IF start THEN
FindAndReplace(pSrcString:= ADR(cmdIn), pDeleteString:= ADR('#1#'), pInsertString:= ADR(GVL_HMI.stRecipeInfo.sMethodName), pDstString:= ADR(cmdIn), nDstSize:= SIZEOF(cmdIn));
FindAndReplace(pSrcString:= ADR(cmdIn), pDeleteString:= ADR('#2#'), pInsertString:= ADR(iRevision), pDstString:= ADR(cmdIn), nDstSize:= SIZEOF(cmdIn));
FindAndReplace(pSrcString:= ADR(cmdIn), pDeleteString:= ADR('#3#'), pInsertString:= ADR(GVL_HMI.stRecipeInfo.sCreatedBy), pDstString:= ADR(cmdIn), nDstSize:= SIZEOF(cmdIn));
FindAndReplace(pSrcString:= ADR(cmdIn), pDeleteString:= ADR('#4#'), pInsertString:= ADR(dCreationDate), pDstString:= ADR(cmdIn), nDstSize:= SIZEOF(cmdIn));
FindAndReplace(pSrcString:= ADR(cmdIn), pDeleteString:= ADR('#5#'), pInsertString:= ADR(Rinse1), pDstString:= ADR(cmdIn), nDstSize:= SIZEOF(cmdIn));
FindAndReplace(pSrcString:= ADR(cmdIn), pDeleteString:= ADR('#6#'), pInsertString:= ADR(Rinse2), pDstString:= ADR(cmdIn), nDstSize:= SIZEOF(cmdIn));
FindAndReplace(pSrcString:= ADR(cmdIn), pDeleteString:= ADR('#7#'), pInsertString:= ADR(Wash1), pDstString:= ADR(cmdIn), nDstSize:= SIZEOF(cmdIn));
FindAndReplace(pSrcString:= ADR(cmdIn), pDeleteString:= ADR('#8#'), pInsertString:= ADR(Wash2), pDstString:= ADR(cmdIn), nDstSize:= SIZEOF(cmdIn));
FindAndReplace(pSrcString:= ADR(cmdIn), pDeleteString:= ADR('#9#'), pInsertString:= ADR(Rinse12), pDstString:= ADR(cmdIn), nDstSize:= SIZEOF(cmdIn));
FindAndReplace(pSrcString:= ADR(cmdIn), pDeleteString:= ADR('#10#'), pInsertString:= ADR(Rinse22), pDstString:= ADR(cmdIn), nDstSize:= SIZEOF(cmdIn));
FindAndReplace(pSrcString:= ADR(cmdIn), pDeleteString:= ADR('#11#'), pInsertString:= ADR(Wash12), pDstString:= ADR(cmdIn), nDstSize:= SIZEOF(cmdIn));
FindAndReplace(pSrcString:= ADR(cmdIn), pDeleteString:= ADR('#12#'), pInsertString:= ADR(Wash22), pDstString:= ADR(cmdIn), nDstSize:= SIZEOF(cmdIn));
FindAndReplace(pSrcString:= ADR(cmdIn), pDeleteString:= ADR('#13#'), pInsertString:= ADR(Rinse13), pDstString:= ADR(cmdIn), nDstSize:= SIZEOF(cmdIn));
FindAndReplace(pSrcString:= ADR(cmdIn), pDeleteString:= ADR('#14#'), pInsertString:= ADR(Rinse23), pDstString:= ADR(cmdIn), nDstSize:= SIZEOF(cmdIn));
FindAndReplace(pSrcString:= ADR(cmdIn), pDeleteString:= ADR('#15#'), pInsertString:= ADR(Wash13), pDstString:= ADR(cmdIn), nDstSize:= SIZEOF(cmdIn));
FindAndReplace(pSrcString:= ADR(cmdIn), pDeleteString:= ADR('#16#'), pInsertString:= ADR(Wash23), pDstString:= ADR(cmdIn), nDstSize:= SIZEOF(cmdIn));
FindAndReplace(pSrcString:= ADR(cmdIn), pDeleteString:= ADR('#17#'), pInsertString:= ADR(soakTime), pDstString:= ADR(cmdIn), nDstSize:= SIZEOF(cmdIn));
FindAndReplace(pSrcString:= ADR(cmdIn), pDeleteString:= ADR('#18#'), pInsertString:= ADR(agitate_1_Time), pDstString:= ADR(cmdIn), nDstSize:= SIZEOF(cmdIn));
FindAndReplace(pSrcString:= ADR(cmdIn), pDeleteString:= ADR('#19#'), pInsertString:= ADR(agitate_2_Time), pDstString:= ADR(cmdIn), nDstSize:= SIZEOF(cmdIn));
FindAndReplace(pSrcString:= ADR(cmdIn), pDeleteString:= ADR('#20#'), pInsertString:= ADR(vialsToFill), pDstString:= ADR(cmdIn), nDstSize:= SIZEOF(cmdIn));
FindAndReplace(pSrcString:= ADR(cmdIn), pDeleteString:= ADR('#21#'), pInsertString:= ADR(vialPrimeVol), pDstString:= ADR(cmdIn), nDstSize:= SIZEOF(cmdIn));
FindAndReplace(pSrcString:= ADR(cmdIn), pDeleteString:= ADR('#22#'), pInsertString:= ADR(vial_1_FillVol), pDstString:= ADR(cmdIn), nDstSize:= SIZEOF(cmdIn));
FindAndReplace(pSrcString:= ADR(cmdIn), pDeleteString:= ADR('#23#'), pInsertString:= ADR(vial_2_4_FillVol), pDstString:= ADR(cmdIn), nDstSize:= SIZEOF(cmdIn));
FindAndReplace(pSrcString:= ADR(cmdIn), pDeleteString:= ADR('#24#'), pInsertString:= ADR(airDryTime), pDstString:= ADR(cmdIn), nDstSize:= SIZEOF(cmdIn));
FindAndReplace(pSrcString:= ADR(cmdIn), pDeleteString:= ADR('#25#'), pInsertString:= ADR('activated'), pDstString:= ADR(cmdIn), nDstSize:= SIZEOF(cmdIn));

END_IF
END_METHOD

METHOD insertRunValues : BOOL
VAR_INPUT
	start: bool;
END_VAR

VAR
	methodID: STRING;
	CalibrationNo: STRING;
END_VAR
methodID:= INT_TO_STRING(GVL_DB.stPostRunInfo.methodID);
CalibrationNo:= INT_TO_STRING(GVL_DB.stPostRunInfo.CalibrationNo);

IF start THEN
FindAndReplace(pSrcString:= ADR(cmdIn), pDeleteString:= ADR('#1#'), pInsertString:= ADR(GVL_DB.stPostRunInfo.analyst), pDstString:= ADR(cmdIn), nDstSize:= SIZEOF(cmdIn));
FindAndReplace(pSrcString:= ADR(cmdIn), pDeleteString:= ADR('#2#'), pInsertString:= ADR(GVL_DB.stPostRunInfo.comment), pDstString:= ADR(cmdIn), nDstSize:= SIZEOF(cmdIn));
FindAndReplace(pSrcString:= ADR(cmdIn), pDeleteString:= ADR('#3#'), pInsertString:= ADR(GVL_DB.stPostRunInfo.softwareVersion), pDstString:= ADR(cmdIn), nDstSize:= SIZEOF(cmdIn));
FindAndReplace(pSrcString:= ADR(cmdIn), pDeleteString:= ADR('#4#'), pInsertString:= ADR(GVL_DB.stPostRunInfo.sysMasterRevision), pDstString:= ADR(cmdIn), nDstSize:= SIZEOF(cmdIn));
FindAndReplace(pSrcString:= ADR(cmdIn), pDeleteString:= ADR('#5#'), pInsertString:= ADR(GVL_DB.stPostRunInfo.sysSettingsRevision), pDstString:= ADR(cmdIn), nDstSize:= SIZEOF(cmdIn));
FindAndReplace(pSrcString:= ADR(cmdIn), pDeleteString:= ADR('#6#'), pInsertString:= ADR(GVL_DB.stPostRunInfo.meterVelocity), pDstString:= ADR(cmdIn), nDstSize:= SIZEOF(cmdIn));
FindAndReplace(pSrcString:= ADR(cmdIn), pDeleteString:= ADR('#7#'), pInsertString:= ADR(GVL_DB.stPostRunInfo.runVelocity), pDstString:= ADR(cmdIn), nDstSize:= SIZEOF(cmdIn));
FindAndReplace(pSrcString:= ADR(cmdIn), pDeleteString:= ADR('#8#'), pInsertString:= ADR(GVL_DB.stPostRunInfo.emptyTubesFactor), pDstString:= ADR(cmdIn), nDstSize:= SIZEOF(cmdIn));
FindAndReplace(pSrcString:= ADR(cmdIn), pDeleteString:= ADR('#9#'), pInsertString:= ADR(GVL_DB.stPostRunInfo.fillTubesFactor), pDstString:= ADR(cmdIn), nDstSize:= SIZEOF(cmdIn));
FindAndReplace(pSrcString:= ADR(cmdIn), pDeleteString:= ADR('#10#'), pInsertString:= ADR(GVL_DB.stPostRunInfo.solvent1NameRevision), pDstString:= ADR(cmdIn), nDstSize:= SIZEOF(cmdIn));
FindAndReplace(pSrcString:= ADR(cmdIn), pDeleteString:= ADR('#11#'), pInsertString:= ADR(GVL_DB.stPostRunInfo.solvent2NameRevision), pDstString:= ADR(cmdIn), nDstSize:= SIZEOF(cmdIn));
FindAndReplace(pSrcString:= ADR(cmdIn), pDeleteString:= ADR('#12#'), pInsertString:= ADR(GVL_DB.stPostRunInfo.solvent3NameRevision), pDstString:= ADR(cmdIn), nDstSize:= SIZEOF(cmdIn));
FindAndReplace(pSrcString:= ADR(cmdIn), pDeleteString:= ADR('#13#'), pInsertString:= ADR(GVL_DB.stPostRunInfo.solvent4NameRevision), pDstString:= ADR(cmdIn), nDstSize:= SIZEOF(cmdIn));
FindAndReplace(pSrcString:= ADR(cmdIn), pDeleteString:= ADR('#14#'), pInsertString:= ADR(GVL_DB.stPostRunInfo.timeEventStarted), pDstString:= ADR(cmdIn), nDstSize:= SIZEOF(cmdIn));
FindAndReplace(pSrcString:= ADR(cmdIn), pDeleteString:= ADR('#15#'), pInsertString:= ADR(GVL_DB.stPostRunInfo.timeEventCompleted), pDstString:= ADR(cmdIn), nDstSize:= SIZEOF(cmdIn));
FindAndReplace(pSrcString:= ADR(cmdIn), pDeleteString:= ADR('#16#'), pInsertString:= ADR(methodID), pDstString:= ADR(cmdIn), nDstSize:= SIZEOF(cmdIn));
FindAndReplace(pSrcString:= ADR(cmdIn), pDeleteString:= ADR('#17#'), pInsertString:= ADR(CalibrationNo), pDstString:= ADR(cmdIn), nDstSize:= SIZEOF(cmdIn));
END_IF
END_METHOD

METHOD insertSolvent : BOOL
VAR_INPUT
	start: BOOL;
END_VAR


VAR

END_VAR


IF start THEN
	FindAndReplace(pSrcString:= ADR(cmdIn), pDeleteString:= ADR('#1#'), pInsertString:= ADR(GVL_DB.stSolvents.solventName1), pDstString:= ADR(cmdIn), nDstSize:= SIZEOF(cmdIn));
	FindAndReplace(pSrcString:= ADR(cmdIn), pDeleteString:= ADR('#2#'), pInsertString:= ADR(GVL_DB.stSolvents.solventName2), pDstString:= ADR(cmdIn), nDstSize:= SIZEOF(cmdIn));
	FindAndReplace(pSrcString:= ADR(cmdIn), pDeleteString:= ADR('#3#'), pInsertString:= ADR(GVL_DB.stSolvents.solventName3), pDstString:= ADR(cmdIn), nDstSize:= SIZEOF(cmdIn));
	FindAndReplace(pSrcString:= ADR(cmdIn), pDeleteString:= ADR('#4#'), pInsertString:= ADR(GVL_DB.stSolvents.solventName4), pDstString:= ADR(cmdIn), nDstSize:= SIZEOF(cmdIn));
	FindAndReplace(pSrcString:= ADR(cmdIn), pDeleteString:= ADR('#5#'), pInsertString:= ADR(GVL_DB.stSolvents.density1), pDstString:= ADR(cmdIn), nDstSize:= SIZEOF(cmdIn));
	FindAndReplace(pSrcString:= ADR(cmdIn), pDeleteString:= ADR('#6#'), pInsertString:= ADR(GVL_DB.stSolvents.density2), pDstString:= ADR(cmdIn), nDstSize:= SIZEOF(cmdIn));
	FindAndReplace(pSrcString:= ADR(cmdIn), pDeleteString:= ADR('#7#'), pInsertString:= ADR(GVL_DB.stSolvents.density3), pDstString:= ADR(cmdIn), nDstSize:= SIZEOF(cmdIn));
	FindAndReplace(pSrcString:= ADR(cmdIn), pDeleteString:= ADR('#8#'), pInsertString:= ADR(GVL_DB.stSolvents.density4), pDstString:= ADR(cmdIn), nDstSize:= SIZEOF(cmdIn));
	FindAndReplace(pSrcString:= ADR(cmdIn), pDeleteString:= ADR('#9#'), pInsertString:= ADR(GVL_DB.stSolvents.addedBy), pDstString:= ADR(cmdIn), nDstSize:= SIZEOF(cmdIn));
	FindAndReplace(pSrcString:= ADR(cmdIn), pDeleteString:= ADR('#10#'), pInsertString:= ADR(GVL_DB.stSolvents.addedDate), pDstString:= ADR(cmdIn), nDstSize:= SIZEOF(cmdIn));
END_IF
END_METHOD

METHOD insertSys : BOOL
VAR_INPUT
	start: BOOL;
END_VAR

VAR
	bGeneralSealAndPump: STRING;
	rAcceptanceCriteria: STRING;
	iAllowableFailures: STRING;
	iReplicatesSetpoint: STRING;
	iCalIntervalDays: STRING;
	iAirDryTimeSec: STRING;
	iAllowableLeakTestFailures: STRING;
	tLeakTestBuildUpTime: STRING;
	tLeakTestMonitorTime: STRING;
	rLeakTestPressureLimit: STRING;
	sealPosition: STRING;
	dryposition: STRING;
	rM1Velocity: STRING;
	iMeterVelocity: STRING;
	iRunVelocity: STRING;
	iEmptyFactor: STRING;
	iFillolventTubesFactor: STRING;
	abovecalibration: STRING;
	vialsetspacing: STRING;
	intoresbottom: STRING;
	intodispense: STRING;
	intoweight: STRING;
	intovials: STRING;
	bDisplayManualControl: STRING;
	bCheckLogonEachRun: STRING;
	abovevialset1: STRING;
	intoWaste: STRING;
	userName: STRING;
	savedDate: STRING;
	
	// Timestamp generation (local system time)
    fbLocalSystemTime : FB_LocalSystemTime;
    stLocal           : TIMESTRUCT;
    sStamp            : STRING(32);
    sHH               : STRING(2);
    sMM               : STRING(2);
    sSS               : STRING(2);
    sMMo              : STRING(3);
    sDD               : STRING(2);
	bDTReady		  : BOOL := FALSE;

END_VAR
bGeneralSealAndPump := BOOL_TO_STRING(GVL_Settings.bGeneralSealAndPump);
rAcceptanceCriteria := LREAL_TO_STRING(GVL_Settings.stCalibParameters.rAcceptanceCriteria);
iAllowableFailures  := USINT_TO_STRING(GVL_Settings.stCalibParameters.iAllowableFailures);
iReplicatesSetpoint := UINT_TO_STRING(GVL_Settings.stCalibParameters.iReplicatesSetpoint);
iCalIntervalDays := UINT_TO_STRING(GVL_Settings.stCalibParameters.iCalIntervalDays);
iAirDryTimeSec := UINT_TO_STRING(GVL_Settings.stCalibParameters.iAirDryTimeSec);
iAllowableLeakTestFailures := UINT_TO_STRING(GVL_Settings.stLeakTestParameters.iAllowableLeakTestFailures);
tLeakTestBuildUpTime := UINT_TO_STRING(GVL_Settings.stLeakTestParameters.tLeakTestBuildUpTime);
tLeakTestMonitorTime := UINT_TO_STRING(GVL_Settings.stLeakTestParameters.tLeakTestMonitorTime);
rLeakTestPressureLimit := REAL_TO_STRING(GVL_Settings.stLeakTestParameters.rLeakTestPressureLimit);
sealPosition := INT_TO_STRING(GVL_Settings.stMachineParam.aM1Position[2]);
dryposition := INT_TO_STRING(GVL_Settings.stMachineParam.aM1Position[3]);
rM1Velocity := LREAL_TO_STRING(GVL_Settings.stMachineParam.rM1Velocity);
iMeterVelocity := UINT_TO_STRING(GVL_Settings.stPumpParameters.iMeterVelocity);
iRunVelocity := UINT_TO_STRING(GVL_Settings.stPumpParameters.iRunVelocity);
iEmptyFactor := UINT_TO_STRING(GVL_Settings.stPumpParameters.iEmptyFactor);
iFillolventTubesFactor := UINT_TO_STRING(GVL_Settings.stPumpParameters.iFillolventTubesFactor);
abovecalibration := INT_TO_STRING(GVL_Settings.stMachineParam.aM3Position[4]);
vialsetspacing := INT_TO_STRING(GVL_Settings.stMachineParam.aM3Position[3]);
intoresbottom := INT_TO_STRING(GVL_Settings.stMachineParam.aM2Position[4]);
intodispense := INT_TO_STRING(GVL_Settings.stMachineParam.aM2Position[5]);
intoweight := INT_TO_STRING(GVL_Settings.stMachineParam.aM2Position[6]);
intovials := INT_TO_STRING(GVL_Settings.stMachineParam.aM2Position[3]);
bDisplayManualControl := BOOL_TO_STRING(GVL_Settings.bDisplayManualControl);
bCheckLogonEachRun := BOOL_TO_STRING(GVL_Settings.bCheckLogonEachRun);
abovevialset1 := INT_TO_STRING(GVL_Settings.stMachineParam.aM3Position[2]);
intoWaste := INT_TO_STRING(GVL_Settings.stMachineParam.aM2Position[2]);
userName := GVL_HMI.sUserNameEventTriggered;
savedDate := GVL_HMI.sDateAndTimeEventTriggered;

IF start THEN
	FindAndReplace(pSrcString:= ADR(cmdIn), pDeleteString:= ADR('#1#'), pInsertString:= ADR(bGeneralSealAndPump), pDstString:= ADR(cmdIn), nDstSize:= SIZEOF(cmdIn));
	FindAndReplace(pSrcString:= ADR(cmdIn), pDeleteString:= ADR('#2#'), pInsertString:= ADR(rAcceptanceCriteria), pDstString:= ADR(cmdIn), nDstSize:= SIZEOF(cmdIn));
	FindAndReplace(pSrcString:= ADR(cmdIn), pDeleteString:= ADR('#3#'), pInsertString:= ADR(iAllowableFailures), pDstString:= ADR(cmdIn), nDstSize:= SIZEOF(cmdIn));
	FindAndReplace(pSrcString:= ADR(cmdIn), pDeleteString:= ADR('#4#'), pInsertString:= ADR(iReplicatesSetpoint), pDstString:= ADR(cmdIn), nDstSize:= SIZEOF(cmdIn));
	FindAndReplace(pSrcString:= ADR(cmdIn), pDeleteString:= ADR('#5#'), pInsertString:= ADR(iCalIntervalDays), pDstString:= ADR(cmdIn), nDstSize:= SIZEOF(cmdIn));
	FindAndReplace(pSrcString:= ADR(cmdIn), pDeleteString:= ADR('#6#'), pInsertString:= ADR('N/A'), pDstString:= ADR(cmdIn), nDstSize:= SIZEOF(cmdIn));
	FindAndReplace(pSrcString:= ADR(cmdIn), pDeleteString:= ADR('#7#'), pInsertString:= ADR(iAirDryTimeSec), pDstString:= ADR(cmdIn), nDstSize:= SIZEOF(cmdIn));
	FindAndReplace(pSrcString:= ADR(cmdIn), pDeleteString:= ADR('#8#'), pInsertString:= ADR(iAllowableLeakTestFailures), pDstString:= ADR(cmdIn), nDstSize:= SIZEOF(cmdIn));
	FindAndReplace(pSrcString:= ADR(cmdIn), pDeleteString:= ADR('#9#'), pInsertString:= ADR(tLeakTestBuildUpTime), pDstString:= ADR(cmdIn), nDstSize:= SIZEOF(cmdIn));
	FindAndReplace(pSrcString:= ADR(cmdIn), pDeleteString:= ADR('#10#'), pInsertString:= ADR(tLeakTestMonitorTime), pDstString:= ADR(cmdIn), nDstSize:= SIZEOF(cmdIn));
	FindAndReplace(pSrcString:= ADR(cmdIn), pDeleteString:= ADR('#11#'), pInsertString:= ADR(rLeakTestPressureLimit), pDstString:= ADR(cmdIn), nDstSize:= SIZEOF(cmdIn));
	FindAndReplace(pSrcString:= ADR(cmdIn), pDeleteString:= ADR('#12#'), pInsertString:= ADR(sealPosition), pDstString:= ADR(cmdIn), nDstSize:= SIZEOF(cmdIn));
	FindAndReplace(pSrcString:= ADR(cmdIn), pDeleteString:= ADR('#13#'), pInsertString:= ADR(dryposition), pDstString:= ADR(cmdIn), nDstSize:= SIZEOF(cmdIn));
	FindAndReplace(pSrcString:= ADR(cmdIn), pDeleteString:= ADR('#14#'), pInsertString:= ADR(rM1Velocity), pDstString:= ADR(cmdIn), nDstSize:= SIZEOF(cmdIn));
	FindAndReplace(pSrcString:= ADR(cmdIn), pDeleteString:= ADR('#15#'), pInsertString:= ADR('N/A'), pDstString:= ADR(cmdIn), nDstSize:= SIZEOF(cmdIn));
	FindAndReplace(pSrcString:= ADR(cmdIn), pDeleteString:= ADR('#16#'), pInsertString:= ADR('N/A'), pDstString:= ADR(cmdIn), nDstSize:= SIZEOF(cmdIn));
	FindAndReplace(pSrcString:= ADR(cmdIn), pDeleteString:= ADR('#17#'), pInsertString:= ADR('N/A'), pDstString:= ADR(cmdIn), nDstSize:= SIZEOF(cmdIn));
	FindAndReplace(pSrcString:= ADR(cmdIn), pDeleteString:= ADR('#18#'), pInsertString:= ADR(iMeterVelocity), pDstString:= ADR(cmdIn), nDstSize:= SIZEOF(cmdIn));
	FindAndReplace(pSrcString:= ADR(cmdIn), pDeleteString:= ADR('#19#'), pInsertString:= ADR(iRunVelocity), pDstString:= ADR(cmdIn), nDstSize:= SIZEOF(cmdIn));
	FindAndReplace(pSrcString:= ADR(cmdIn), pDeleteString:= ADR('#20#'), pInsertString:= ADR(iEmptyFactor), pDstString:= ADR(cmdIn), nDstSize:= SIZEOF(cmdIn));
	FindAndReplace(pSrcString:= ADR(cmdIn), pDeleteString:= ADR('#21#'), pInsertString:= ADR(iFillolventTubesFactor), pDstString:= ADR(cmdIn), nDstSize:= SIZEOF(cmdIn));
	FindAndReplace(pSrcString:= ADR(cmdIn), pDeleteString:= ADR('#22#'), pInsertString:= ADR(abovecalibration), pDstString:= ADR(cmdIn), nDstSize:= SIZEOF(cmdIn));
	FindAndReplace(pSrcString:= ADR(cmdIn), pDeleteString:= ADR('#23#'), pInsertString:= ADR(vialsetspacing), pDstString:= ADR(cmdIn), nDstSize:= SIZEOF(cmdIn));
	FindAndReplace(pSrcString:= ADR(cmdIn), pDeleteString:= ADR('#24#'), pInsertString:= ADR(intoresbottom), pDstString:= ADR(cmdIn), nDstSize:= SIZEOF(cmdIn));
	FindAndReplace(pSrcString:= ADR(cmdIn), pDeleteString:= ADR('#25#'), pInsertString:= ADR(intodispense), pDstString:= ADR(cmdIn), nDstSize:= SIZEOF(cmdIn));
	FindAndReplace(pSrcString:= ADR(cmdIn), pDeleteString:= ADR('#26#'), pInsertString:= ADR(intoweight), pDstString:= ADR(cmdIn), nDstSize:= SIZEOF(cmdIn));
	FindAndReplace(pSrcString:= ADR(cmdIn), pDeleteString:= ADR('#27#'), pInsertString:= ADR(intovials), pDstString:= ADR(cmdIn), nDstSize:= SIZEOF(cmdIn));
	FindAndReplace(pSrcString:= ADR(cmdIn), pDeleteString:= ADR('#28#'), pInsertString:= ADR(bDisplayManualControl), pDstString:= ADR(cmdIn), nDstSize:= SIZEOF(cmdIn));
	FindAndReplace(pSrcString:= ADR(cmdIn), pDeleteString:= ADR('#29#'), pInsertString:= ADR(bCheckLogonEachRun), pDstString:= ADR(cmdIn), nDstSize:= SIZEOF(cmdIn));
	FindAndReplace(pSrcString:= ADR(cmdIn), pDeleteString:= ADR('#30#'), pInsertString:= ADR(userName), pDstString:= ADR(cmdIn), nDstSize:= SIZEOF(cmdIn));
	FindAndReplace(pSrcString:= ADR(cmdIn), pDeleteString:= ADR('#31#'), pInsertString:= ADR(savedDate), pDstString:= ADR(cmdIn), nDstSize:= SIZEOF(cmdIn));
	FindAndReplace(pSrcString:= ADR(cmdIn), pDeleteString:= ADR('#32#'), pInsertString:= ADR(abovevialset1), pDstString:= ADR(cmdIn), nDstSize:= SIZEOF(cmdIn));
	FindAndReplace(pSrcString:= ADR(cmdIn), pDeleteString:= ADR('#33#'), pInsertString:= ADR(intoWaste), pDstString:= ADR(cmdIn), nDstSize:= SIZEOF(cmdIn));
END_IF
END_METHOD

METHOD insertUser : BOOL
VAR_INPUT
	start: BOOL;
	line: INT;
END_VAR


IF start THEN
	FindAndReplace(pSrcString:= ADR(cmdIn), pDeleteString:= ADR('#1#'), pInsertString:= ADR(GVL_DB.astData_CUL[line].userID), pDstString:= ADR(cmdIn), nDstSize:= SIZEOF(cmdIn));
	FindAndReplace(pSrcString:= ADR(cmdIn), pDeleteString:= ADR('#2#'), pInsertString:= ADR(GVL_DB.astData_CUL[line].acessLevel), pDstString:= ADR(cmdIn), nDstSize:= SIZEOF(cmdIn));
	FindAndReplace(pSrcString:= ADR(cmdIn), pDeleteString:= ADR('#3#'), pInsertString:= ADR(GVL_DB.astData_CUL[line].transactionType), pDstString:= ADR(cmdIn), nDstSize:= SIZEOF(cmdIn));
	FindAndReplace(pSrcString:= ADR(cmdIn), pDeleteString:= ADR('#4#'), pInsertString:= ADR(GVL_DB.astData_CUL[line].transactionDate), pDstString:= ADR(cmdIn), nDstSize:= SIZEOF(cmdIn));
	FindAndReplace(pSrcString:= ADR(cmdIn), pDeleteString:= ADR('#5#'), pInsertString:= ADR(GVL_DB.astData_CUL[line].transactedBy), pDstString:= ADR(cmdIn), nDstSize:= SIZEOF(cmdIn));
	FindAndReplace(pSrcString:= ADR(cmdIn), pDeleteString:= ADR('#6#'), pInsertString:= ADR(GVL_DB.astData_CUL[line].addDate), pDstString:= ADR(cmdIn), nDstSize:= SIZEOF(cmdIn));
	FindAndReplace(pSrcString:= ADR(cmdIn), pDeleteString:= ADR('#7#'), pInsertString:= ADR(GVL_DB.astData_CUL[line].enteredBy), pDstString:= ADR(cmdIn), nDstSize:= SIZEOF(cmdIn));
END_IF
END_METHOD

METHOD insertUserMgmtHistory : BOOL
VAR_INPUT
	start : BOOL := FALSE;
END_VAR
VAR
    sOldAutoLogoutMin : STRING(20);
    sNewAutoLogoutMin : STRING(20);
END_VAR
sOldAutoLogoutMin := INT_TO_STRING(GVL_HMI.stUserMgmtHistoryEvent.iOldAutoLogoutMin);
sNewAutoLogoutMin := INT_TO_STRING(GVL_HMI.stUserMgmtHistoryEvent.iNewAutoLogoutMin);

IF start THEN

    FindAndReplace(
        pSrcString := ADR(cmdIn), 
        pDeleteString := ADR('#1#'), 
        pInsertString := ADR(GVL_HMI.stUserMgmtHistoryEvent.sTargetUser), 
        pDstString := ADR(cmdIn), 
        nDstSize := SIZEOF(cmdIn)
    );

    FindAndReplace(
        pSrcString := ADR(cmdIn), 
        pDeleteString := ADR('#2#'), 
        pInsertString := ADR(GVL_HMI.stUserMgmtHistoryEvent.sEventType), 
        pDstString := ADR(cmdIn), 
        nDstSize := SIZEOF(cmdIn)
    );

    FindAndReplace(
        pSrcString := ADR(cmdIn), 
        pDeleteString := ADR('#3#'), 
        pInsertString := ADR(GVL_HMI.stUserMgmtHistoryEvent.sOldGroup), 
        pDstString := ADR(cmdIn), 
        nDstSize := SIZEOF(cmdIn)
    );

    FindAndReplace(
        pSrcString := ADR(cmdIn), 
        pDeleteString := ADR('#4#'), 
        pInsertString := ADR(GVL_HMI.stUserMgmtHistoryEvent.sNewGroup), 
        pDstString := ADR(cmdIn), 
        nDstSize := SIZEOF(cmdIn)
    );

    FindAndReplace(
        pSrcString := ADR(cmdIn), 
        pDeleteString := ADR('#5#'), 
        pInsertString := ADR(sOldAutoLogoutMin), 
        pDstString := ADR(cmdIn), 
        nDstSize := SIZEOF(cmdIn)
    );

    FindAndReplace(
        pSrcString := ADR(cmdIn), 
        pDeleteString := ADR('#6#'), 
        pInsertString := ADR(sNewAutoLogoutMin), 
        pDstString := ADR(cmdIn), 
        nDstSize := SIZEOF(cmdIn)
    );

    FindAndReplace(
        pSrcString := ADR(cmdIn), 
        pDeleteString := ADR('#7#'), 
        pInsertString := ADR(GVL_HMI.stUserMgmtHistoryEvent.sPerformedBy), 
        pDstString := ADR(cmdIn), 
        nDstSize := SIZEOF(cmdIn)
    );

    FindAndReplace(
        pSrcString := ADR(cmdIn), 
        pDeleteString := ADR('#8#'), 
        pInsertString := ADR(GVL_HMI.stUserMgmtHistoryEvent.sSourceScreen), 
        pDstString := ADR(cmdIn), 
        nDstSize := SIZEOF(cmdIn)
    );

    FindAndReplace(
        pSrcString := ADR(cmdIn), 
        pDeleteString := ADR('#9#'), 
        pInsertString := ADR(GVL_HMI.stUserMgmtHistoryEvent.sEventComment), 
        pDstString := ADR(cmdIn), 
        nDstSize := SIZEOF(cmdIn)
    );

END_IF
END_METHOD

METHOD insertVD : BOOL
VAR_INPUT
	start: BOOL;
	methodID: STRING;
	line: INT;
END_VAR


VAR
	sysRevisionNo: STRING;
END_VAR


IF start THEN
	FindAndReplace(pSrcString:= ADR(cmdIn), pDeleteString:= ADR('#1#'), pInsertString:= ADR(GVL_DB.astVolData[line].pump), pDstString:= ADR(cmdIn), nDstSize:= SIZEOF(cmdIn));
	FindAndReplace(pSrcString:= ADR(cmdIn), pDeleteString:= ADR('#2#'), pInsertString:= ADR(GVL_DB.astVolData[line].stage), pDstString:= ADR(cmdIn), nDstSize:= SIZEOF(cmdIn));
	FindAndReplace(pSrcString:= ADR(cmdIn), pDeleteString:= ADR('#3#'), pInsertString:= ADR(GVL_DB.astVolData[line].rinse1), pDstString:= ADR(cmdIn), nDstSize:= SIZEOF(cmdIn));
	FindAndReplace(pSrcString:= ADR(cmdIn), pDeleteString:= ADR('#4#'), pInsertString:= ADR(GVL_DB.astVolData[line].rinse2), pDstString:= ADR(cmdIn), nDstSize:= SIZEOF(cmdIn));
	FindAndReplace(pSrcString:= ADR(cmdIn), pDeleteString:= ADR('#5#'), pInsertString:= ADR(GVL_DB.astVolData[line].wash1), pDstString:= ADR(cmdIn), nDstSize:= SIZEOF(cmdIn));
	FindAndReplace(pSrcString:= ADR(cmdIn), pDeleteString:= ADR('#6#'), pInsertString:= ADR(GVL_DB.astVolData[line].wash2), pDstString:= ADR(cmdIn), nDstSize:= SIZEOF(cmdIn));
	FindAndReplace(pSrcString:= ADR(cmdIn), pDeleteString:= ADR('#7#'), pInsertString:= ADR(methodID), pDstString:= ADR(cmdIn), nDstSize:= SIZEOF(cmdIn));
END_IF
END_METHOD

METHOD selectCalibHeader : BOOL
VAR_INPUT
	start : BOOL;
    calibrationNo : STRING;
END_VAR
IF start THEN
    FindAndReplace(
        pSrcString := ADR(cmdSlc),
        pDeleteString := ADR('#1#'),
        pInsertString := ADR(calibrationNo),
        pDstString := ADR(cmdSlc),
        nDstSize := SIZEOF(cmdSlc)
    );
END_IF
END_METHOD

METHOD selectCalibReportHeaderByID : BOOL
VAR_INPUT
	start         : BOOL;
    calibrationID : STRING;
END_VAR
IF start THEN
    Clear_PumpCalibReportBuffers();
    cmdSlc := GVL_DB.slctPumpCalibHeaderByNo1;

    FindAndReplace(
        pSrcString:= ADR(cmdSlc),
        pDeleteString:= ADR('#1#'),
        pInsertString:= ADR(calibrationID),
        pDstString:= ADR(cmdSlc),
        nDstSize:= SIZEOF(cmdSlc)
    );
END_IF
END_METHOD

METHOD selectCalibReportListByDate : BOOL
VAR_INPUT
	start    : BOOL;
    dateFrom : STRING;
    dateTo   : STRING;
END_VAR
IF start THEN
    cmdSlc := GVL_DB.slctCalibReportListByDate;

    FindAndReplace(
        pSrcString    := ADR(cmdSlc),
        pDeleteString := ADR('#1#'),
        pInsertString := ADR(dateFrom),
        pDstString    := ADR(cmdSlc),
        nDstSize      := SIZEOF(cmdSlc)
    );

    FindAndReplace(
        pSrcString    := ADR(cmdSlc),
        pDeleteString := ADR('#2#'),
        pInsertString := ADR(dateTo),
        pDstString    := ADR(cmdSlc),
        nDstSize      := SIZEOF(cmdSlc)
    );
END_IF
END_METHOD

METHOD selectCalibReportValuesByID : BOOL
VAR_INPUT
	start         : BOOL;
    calibrationID : STRING;
END_VAR
IF start THEN
    cmdSlc := GVL_DB.slctPumpCalibValuesByNo1;

    FindAndReplace(
        pSrcString:= ADR(cmdSlc),
        pDeleteString:= ADR('#1#'),
        pInsertString:= ADR(calibrationID),
        pDstString:= ADR(cmdSlc),
        nDstSize:= SIZEOF(cmdSlc)
    );
END_IF
END_METHOD

METHOD selectLinearByID : BOOL
VAR_INPUT
	start    : BOOL;
    linearID : STRING;
END_VAR
IF start THEN
    IF linearID = '' THEN
        cmdSlc := '';
        RETURN;
    END_IF

    cmdSlc := GVL_DB.slctLinearByID;

    FindAndReplace(
        pSrcString := ADR(cmdSlc),
        pDeleteString := ADR('#1#'),
        pInsertString := ADR(linearID),
        pDstString := ADR(cmdSlc),
        nDstSize := SIZEOF(cmdSlc)
    );
END_IF
END_METHOD

METHOD selectLinearReportSearchByDate : BOOL
VAR_INPUT
	start    : BOOL;
    dateFrom : STRING;
    dateTo   : STRING;
END_VAR
IF start THEN
    cmdSlc := GVL_DB.slctLinearReportListByDate;

    FindAndReplace(
        pSrcString := ADR(cmdSlc),
        pDeleteString := ADR('#1#'),
        pInsertString := ADR(dateFrom),
        pDstString := ADR(cmdSlc),
        nDstSize := SIZEOF(cmdSlc)
    );

    FindAndReplace(
        pSrcString := ADR(cmdSlc),
        pDeleteString := ADR('#2#'),
        pInsertString := ADR(dateTo),
        pDstString := ADR(cmdSlc),
        nDstSize := SIZEOF(cmdSlc)
    );
END_IF
END_METHOD

METHOD selectMethod : BOOL
VAR_INPUT
	start: BOOL;
	methodName: STRING;
	methodRevision: STRING;
END_VAR

IF start THEN
FindAndReplace(pSrcString:= ADR(cmdSlc), pDeleteString:= ADR('#1#'), pInsertString:= ADR(methodName), pDstString:= ADR(cmdSlc), nDstSize:= SIZEOF(cmdSlc));
FindAndReplace(pSrcString:= ADR(cmdSlc), pDeleteString:= ADR('#2#'), pInsertString:= ADR(methodRevision), pDstString:= ADR(cmdSlc), nDstSize:= SIZEOF(cmdSlc));
END_IF
END_METHOD

METHOD selectMethodID : BOOL
VAR_INPUT
	start: BOOL;
	methodName: STRING;
END_VAR

IF start THEN
FindAndReplace(pSrcString:= ADR(cmdSlc), pDeleteString:= ADR('#1#'), pInsertString:= ADR(methodName), pDstString:= ADR(cmdSlc), nDstSize:= SIZEOF(cmdSlc));
END_IF
END_METHOD

METHOD selectMethodReportSearchByDate : BOOL
VAR_INPUT
	start    : BOOL;
	dateFrom : STRING;
	dateTo   : STRING;
END_VAR
// Builds the date-filtered method report search query (latest revision per method).
// Replaces #1# with dateFrom and #2# with dateTo.
IF start THEN
    cmdSlc := GVL_DB.slctMethodReportSearchLatestByDate;

    FindAndReplace(
        pSrcString    := ADR(cmdSlc),
        pDeleteString := ADR('#1#'),
        pInsertString := ADR(dateFrom),
        pDstString    := ADR(cmdSlc),
        nDstSize      := SIZEOF(cmdSlc)
    );

    FindAndReplace(
        pSrcString    := ADR(cmdSlc),
        pDeleteString := ADR('#2#'),
        pInsertString := ADR(dateTo),
        pDstString    := ADR(cmdSlc),
        nDstSize      := SIZEOF(cmdSlc)
    );
END_IF
END_METHOD

METHOD selectPostRunHeaderByID : BOOL
VAR_INPUT
	start : BOOL;
    runID : STRING;
END_VAR
IF start THEN
    cmdSlc := GVL_DB.slctPostRunHeaderByID;

    FindAndReplace(
        pSrcString := ADR(cmdSlc),
        pDeleteString := ADR('#1#'),
        pInsertString := ADR(runID),
        pDstString := ADR(cmdSlc),
        nDstSize := SIZEOF(cmdSlc)
    );
END_IF
END_METHOD

METHOD selectPostRunMethodHeaderByID : BOOL
VAR_INPUT
	start    : BOOL;
    methodID : STRING;
END_VAR
IF start THEN
    cmdSlc := GVL_DB.slctPostRunMethodHeaderByID;

    FindAndReplace(
        pSrcString := ADR(cmdSlc),
        pDeleteString := ADR('#1#'),
        pInsertString := ADR(methodID),
        pDstString := ADR(cmdSlc),
        nDstSize := SIZEOF(cmdSlc)
    );
END_IF
END_METHOD

METHOD selectPostRunVolumeByMethodID : BOOL
VAR_INPUT
	start    : BOOL;
    methodID : STRING;
END_VAR
IF start THEN
    cmdSlc := GVL_DB.slctPostRunVolumeByMethodID;

    FindAndReplace(
        pSrcString := ADR(cmdSlc),
        pDeleteString := ADR('#1#'),
        pInsertString := ADR(methodID),
        pDstString := ADR(cmdSlc),
        nDstSize := SIZEOF(cmdSlc)
    );
END_IF
END_METHOD

METHOD selectRecipeHeaderByID : BOOL
VAR_INPUT
	start    : BOOL;
    methodID : STRING;
END_VAR
IF start THEN
    cmdSlc := GVL_DB.slctMethodHeaderByID;

    FindAndReplace(
        pSrcString := ADR(cmdSlc),
        pDeleteString := ADR('#1#'),
        pInsertString := ADR(methodID),
        pDstString := ADR(cmdSlc),
        nDstSize := SIZEOF(cmdSlc)
    );
END_IF
END_METHOD

METHOD selectRecipeVolumeByID : BOOL
VAR_INPUT
	start    : BOOL;
    methodID : STRING;
END_VAR
IF start THEN
    cmdSlc := GVL_DB.slctMethodVolumeByID;

    FindAndReplace(
        pSrcString := ADR(cmdSlc),
        pDeleteString := ADR('#1#'),
        pInsertString := ADR(methodID),
        pDstString := ADR(cmdSlc),
        nDstSize := SIZEOF(cmdSlc)
    );
END_IF
END_METHOD

METHOD selectSystemSettingsByID : BOOL
VAR_INPUT
	start      : BOOL;
    revisionID : STRING;
END_VAR
IF start THEN
    cmdSlc := GVL_DB.slctSystemSettingsByRevision;

    FindAndReplace(
        pSrcString    := ADR(cmdSlc),
        pDeleteString := ADR('#1#'),
        pInsertString := ADR(revisionID),
        pDstString    := ADR(cmdSlc),
        nDstSize      := SIZEOF(cmdSlc)
    );
END_IF
END_METHOD

METHOD selectSystemSettingsReportLisT : BOOL
VAR_INPUT
	start : BOOL;
END_VAR
IF start THEN
    cmdSlc := GVL_DB.slctSystemSettingsReportList;
END_IF
END_METHOD

METHOD selectSystemSettingsReportListByDate : BOOL
VAR_INPUT
	start    : BOOL;
    dateFrom : STRING;
    dateTo   : STRING;
END_VAR
IF start THEN
    cmdSlc := GVL_DB.slctSystemSettingsReportListByDate;

    FindAndReplace(
        pSrcString    := ADR(cmdSlc),
        pDeleteString := ADR('#1#'),
        pInsertString := ADR(dateFrom),
        pDstString    := ADR(cmdSlc),
        nDstSize      := SIZEOF(cmdSlc)
    );

    FindAndReplace(
        pSrcString    := ADR(cmdSlc),
        pDeleteString := ADR('#2#'),
        pInsertString := ADR(dateTo),
        pDstString    := ADR(cmdSlc),
        nDstSize      := SIZEOF(cmdSlc)
    );
END_IF
END_METHOD

METHOD selectVD : BOOL
VAR_INPUT
	start: BOOL;
	methodID: STRING;
END_VAR

IF start THEN
FindAndReplace(pSrcString:= ADR(cmdSlc), pDeleteString:= ADR('#1#'), pInsertString:= ADR(methodID), pDstString:= ADR(cmdSlc), nDstSize:= SIZEOF(cmdSlc));
END_IF
END_METHOD

METHOD updateMethod : BOOL
VAR_INPUT
	start: BOOL;
	methodName: STRING;
	methodRevision: STRING;
END_VAR

IF start THEN
FindAndReplace(pSrcString:= ADR(cmdIn), pDeleteString:= ADR('#1#'), pInsertString:= ADR(methodName), pDstString:= ADR(cmdIn), nDstSize:= SIZEOF(cmdIn));
FindAndReplace(pSrcString:= ADR(cmdIn), pDeleteString:= ADR('#2#'), pInsertString:= ADR(methodRevision), pDstString:= ADR(cmdIn), nDstSize:= SIZEOF(cmdIn));
END_IF
END_METHOD

END_PROGRAM

// ---- POUs/MARCO/DB/DB_Load_CompleteMethod.TcPOU
PROGRAM DB_Load_CompleteMethod
VAR
	state: INT;
	timer: ton;
	timer2: ton;
	rev: INT := 1;
	x: INT;
END_VAR

VAR_IN_OUT
	start: BOOL;
END_VAR

timer();
timer2();

CASE state OF
	
0:
	IF start THEN
		DB_Query.state:= E_DB_QUERY_STATE.SELECT_WHOLE_METHODS;
		timer(in:=TRUE, pt:=T#1S);
		state:= 10;
	ELSE
		state:= 0;
	END_IF
	
10:

	IF NOT DB_Query.FB_SelectArray.bBusy AND timer.Q THEN
		//start:= TRUE;	
		timer(in:=FALSE);
		GVL_DB.arrCompleteMethod[rev].agitate_1_Time := GVL_DB.stParameter_MR.agitate_1_Time;
		GVL_DB.arrCompleteMethod[rev].agitate_2_Time := GVL_DB.stParameter_MR.agitate_2_Time;
		GVL_DB.arrCompleteMethod[rev].airDryTime := GVL_DB.stParameter_MR.airDryTime;
		GVL_DB.arrCompleteMethod[rev].methodCreatedBy := GVL_DB.stParameter_MR.methodCreatedBy;
		GVL_DB.arrCompleteMethod[rev].methodCreatedOn := GVL_DB.stParameter_MR.methodCreatedOn;
		GVL_DB.arrCompleteMethod[rev].methodID := GVL_DB.stParameter_MR.methodID;
		GVL_DB.arrCompleteMethod[rev].methodName := GVL_DB.stParameter_MR.methodName;
		GVL_DB.arrCompleteMethod[rev].methodRevision := GVL_DB.stParameter_MR.methodRevision;
		GVL_DB.arrCompleteMethod[rev].methodStatus := GVL_DB.stParameter_MR.methodStatus;
		GVL_DB.arrCompleteMethod[rev].soakTime := GVL_DB.stParameter_MR.soakTime;
		GVL_DB.arrCompleteMethod[rev].solvent_R1 := GVL_DB.stParameter_MR.solvent_R1;
		GVL_DB.arrCompleteMethod[rev].solvent_R2 := GVL_DB.stParameter_MR.solvent_R2;
		GVL_DB.arrCompleteMethod[rev].solvent_W1 := GVL_DB.stParameter_MR.solvent_W1;
		GVL_DB.arrCompleteMethod[rev].solvent_W2 := GVL_DB.stParameter_MR.solvent_W2;
		GVL_DB.arrCompleteMethod[rev].time_R1 := GVL_DB.stParameter_MR.time_R1;
		GVL_DB.arrCompleteMethod[rev].time_R2 := GVL_DB.stParameter_MR.time_R2;
		GVL_DB.arrCompleteMethod[rev].time_W1 := GVL_DB.stParameter_MR.time_W1;
		GVL_DB.arrCompleteMethod[rev].time_W2 := GVL_DB.stParameter_MR.time_W2;
		GVL_DB.arrCompleteMethod[rev].velocity_R1 := GVL_DB.stParameter_MR.velocity_R1;
		GVL_DB.arrCompleteMethod[rev].velocity_R2 := GVL_DB.stParameter_MR.velocity_R2;
		GVL_DB.arrCompleteMethod[rev].velocity_W1 := GVL_DB.stParameter_MR.velocity_W1;
		GVL_DB.arrCompleteMethod[rev].velocity_W2 := GVL_DB.stParameter_MR.velocity_W2;
		GVL_DB.arrCompleteMethod[rev].vial_1_FillVol := GVL_DB.stParameter_MR.vial_1_FillVol;
		GVL_DB.arrCompleteMethod[rev].vial_2_4_FillVol := GVL_DB.stParameter_MR.vial_2_4_FillVol;
		GVL_DB.arrCompleteMethod[rev].vialPrimeVol := GVL_DB.stParameter_MR.vialPrimeVol;
		GVL_DB.arrCompleteMethod[rev].vialsToFill := GVL_DB.stParameter_MR.vialsToFill;
		//DB_Query.state:= E_DB_QUERY_STATE.SELECT_VOLUME_DATA;
		timer2(in:= TRUE, pt:= T#5S);
		
		state:= 20;
	ELSE
		state:= 10;
	END_IF
	
20:

	IF NOT DB_Query.FB_SelectArray.bBusy AND timer2.Q THEN
		timer2(in:= FALSE);
		FOR x:= 1 TO 10 BY 1 DO
			GVL_DB.arrCompleteMethod[rev].volumeData[x].pump := GVL_DB.astVolData[x].pump;
			GVL_DB.arrCompleteMethod[rev].volumeData[x].rinse1 := GVL_DB.astVolData[x].rinse1;
			GVL_DB.arrCompleteMethod[rev].volumeData[x].rinse2 := GVL_DB.astVolData[x].rinse2;
			GVL_DB.arrCompleteMethod[rev].volumeData[x].stage := GVL_DB.astVolData[x].stage;
			GVL_DB.arrCompleteMethod[rev].volumeData[x].wash1 := GVL_DB.astVolData[x].wash1;
			GVL_DB.arrCompleteMethod[rev].volumeData[x].wash2 := GVL_DB.astVolData[x].wash2;
			GVL_DB.arrCompleteMethod[rev].volumeData[x].VD_ID := GVL_DB.astVolData[x].VD_ID;
			GVL_DB.arrCompleteMethod[rev].volumeData[x].methodID := GVL_DB.astVolData[x].methodID;
		END_FOR
		DB_Query.state:= E_DB_QUERY_STATE.SELECT_WHOLE_METHODS;
		state:= 30;
	ELSE
		state:= 20;
	END_IF

30:
	IF STRING_TO_INT(GVL_DB.methodRevision) > 1	THEN
		rev:= rev +1;
		GVL_DB.methodRevision:= INT_TO_STRING(STRING_TO_INT(GVL_DB.methodRevision) - 1);
		state:= 0;
	ELSIF STRING_TO_INT(GVL_DB.methodRevision) <= 1 THEN
		start:= FALSE;
		timer(in:= TRUE, pt:= T#5S);
		state:= 40;
	ELSE
		state:= 30;
	END_IF
	
40:
	IF timer.Q THEN
		timer(in:=FALSE);
		rev:= 1;
		state:= 0;
	ELSE
		state:= 40;
	END_IF
END_CASE

END_PROGRAM

// ---- POUs/1. MachineControl/PRG_MasterControl.TcPOU
PROGRAM PRG_MasterControl
VAR
	eMachineModePrev 	: E_MachineMode := E_MachineMode.STOPPED;
	bModeChanged	 	: BOOL := FALSE;
	bResetStateMachine	: BOOL := FALSE;
	bResetSMDone		: BOOL := FALSE;
	bStoppedResetDone	: BOOL := FALSE;
	
	//Triggers
	rTriggerStopButton	: R_TRIG;
	rTriggerStartButton	: R_TRIG;
	
	//PowerUp Variables
	tonPowerUp				: ton;
	bPowerUpTimerComplete	: BOOL := FALSE;
	bPowerUpDone			: BOOL := FALSE;
	
	//System Initializing Variables
	tonSystemInitialize		: ton;
	rTrigEnterSystemInit 	: R_TRIG;
	bInitResetStarted    	: BOOL := FALSE;
    bInitResetCompleted  	: BOOL := FALSE;
	bSystemInitTimerStart	: BOOL := FALSE;
	bSystemInitReseted		: BOOL := FALSE;

END_VAR

// =====================================================================================================================
// 0) System Power Up Timer
// =====================================================================================================================
tonPowerUp( IN 	:= TRUE, 
			PT 	:= T#2S,	
			Q 	=> bPowerUpTimerComplete);

IF bPowerUpTimerComplete AND NOT bPowerUpDone THEN
	GVL_HMI.eMachineMode := E_MachineMode.STOPPED;
	bPowerUpDone := TRUE; // Indicates que the initialization is already happened
END_IF

// =====================================================================================================================
// 1) Peripherals monitoring
// =====================================================================================================================

// Mode Change Monitoring
bModeChanged := (GVL_HMI.eMachineMode <> eMachineModePrev);
eMachineModePrev := GVL_HMI.eMachineMode;

// Buttons Triggers
rTriggerStartButton(CLK := GVL_IO.gDigInputs.bStartButton);
rTriggerStopButton(CLK := GVL_IO.gDigInputs.bStopButton);

//Reset Button Blinking
IF (GVL_HMI.eMachineMode = E_MachineMode.IMEDIATE_FAULT) AND NOT GVL_Safety. bSafetyEnable THEN
	GVL_IO.gDigOutputs.bResetIndicator := GVL_Safety.bResetButtonBlink;
END_IF

// Stop Button monitoring
ACT_StopMonitoring();
(*
IF rTriggerStopButton.Q AND NOT (GVL_HMI.eMachineMode = E_MachineMode.SYSTEM_INITIALIZING) THEN
	GVL_HMI.eMachineMode := E_MachineMode.STOPPED;
END_IF
*)

//Safety Enable Monitoring
IF NOT GVL_Safety.bSafetyEnable THEN
	GVL_HMI.eMachineMode := E_MachineMode.IMEDIATE_FAULT;
END_IF

//Reset PRG`s when in system init 
IF (GVL_HMI.eMachineMode = E_MachineMode.SYSTEM_INITIALIZING) THEN
	//PRG_Calibration.Reset();
	PRG_AutoCycle.Reset();
END_IF

//Reset the Reset flags every time gets out of auto cycle
IF NOT (GVL_HMI.eMachineMode = E_MachineMode.AUTO_CYCLE) THEN
	bResetSMDone := FALSE;
	bResetStateMachine := TRUE;
END_IF

//Resets PRG_SystemIniti *********************************************************************************************

IF (GVL_HMI.eMachineMode <> E_MachineMode.SYSTEM_INITIALIZING) AND NOT bSystemInitReseted THEN
	bSystemInitReseted := PRG_SystemInit.Reset();
	IF bSystemInitReseted THEN
		bSystemInitTimerStart := FALSE; //Reset timer every time is not in System Initializing
	END_IF
END_IF
//**********************************************************************************************************************

//Reset the Stopped state flags every time gets out of Stopped State
IF NOT (GVL_HMI.eMachineMode = E_MachineMode.STOPPED) THEN
	bStoppedResetDone := PRG_StoppedState.Reset();
END_IF

// =====================================================================================================================
// 2) Main Master controll logic
// =====================================================================================================================

CASE GVL_HMI.eMachineMode OF

    E_MachineMode.AUTO_CYCLE: 	// Entry from Stopped state
		IF bResetStateMachine THEN
			bResetSMDone := PRG_AutoCycle.Reset(); //Resets the state machine everytime entry this case
		END_IF; 
		
		IF bResetSMDone THEN
			bResetStateMachine := FALSE;
    		PRG_AutoCycle(); // calls the state machine
		END_IF

    E_MachineMode.MANUAL:		// Entry from HMI Selection
        PRG_ManualControl(); 

    E_MachineMode.CALIBRATION:	// Entry from HMI Selection
        PRG_Calibration();

        IF PRG_Calibration.bCalibrationFinished THEN
            GVL_HMI.eMachineMode := E_MachineMode.STOPPED;
			PRG_Calibration.Reset();
        END_IF

    E_MachineMode.IMEDIATE_FAULT: //Entry from Safety Monitoring
        //PRG_SafetyHandle();
        IF GVL_Safety.bSafetyEnable THEN
            GVL_HMI.eMachineMode := E_MachineMode.SYSTEM_INITIALIZING;
        END_IF

    E_MachineMode.STOPPED:		// Entry from Stop Button or Imediate Fault
        IF bStoppedResetDone THEN
			PRG_StoppedState();
		END_IF
		
        IF rTriggerStartButton.Q AND GVL_Safety.bSafetyEnable THEN //only change the state if all motors were stopped
			bStoppedResetDone := FALSE;
            GVL_HMI.eMachineMode := E_MachineMode.SYSTEM_INITIALIZING;
        END_IF
	
	E_MachineMode.SYSTEM_INITIALIZING: // Entry when the machine is first power up to do the homing of the motors
	
       	tonSystemInitialize(IN := bSystemInitTimerStart, PT := T#2S);
		
		bSystemInitReseted := FALSE;
		bSystemInitTimerStart := TRUE;
		
		IF GVL_Safety.bSafetyEnable AND tonSystemInitialize.Q THEN
			PRG_SystemInit(); // Run init procedure
		END_IF
		// Transition to SYSTEM_READY when initialization completes
		IF PRG_SystemInit.bDone AND tonSystemInitialize.Q THEN
			GVL_HMI.eMachineMode := E_MachineMode.SYSTEM_READY;
		END_IF
		
	E_MachineMode.SYSTEM_READY:	// Entry when the start button was pressed on Stop State.
	
		// System Ready housekeeping
        PRG_SystemReady();

        // Changing state condition
        IF GVL_HMI.bSystemReady_ReqAutoCycle THEN
            
            GVL_HMI.bSystemReady_ReqAutoCycle := FALSE;			// Resets the flag
            GVL_HMI.eMachineMode := E_MachineMode.AUTO_CYCLE;	// Change state
        END_IF
		
END_CASE

ACTION ACT_StopMonitoring:
// Stop Button monitoring
IF rTriggerStopButton.Q AND NOT (GVL_HMI.eMachineMode = E_MachineMode.SYSTEM_INITIALIZING) THEN
    
    CASE GVL_HMI.eMachineMode OF

        // --------------------------------------------------------------------
        // AUTO_CYCLE: 1st STOP -> soft hold request
        //             2nd STOP while on hold -> hard STOP
        // --------------------------------------------------------------------
        E_MachineMode.AUTO_CYCLE:
            IF NOT GVL_HMI.bAutoCycleHoldActive THEN
                // First STOP press during Auto Cycle:
                // request a soft hold; PRG_StateMachine
                // will move to PAUSE_STATE at a safe boundary.
                GVL_HMI.bAutoCycleHoldReq 	:= TRUE;
				GVL_HMI.bAutoCycleHoldPopup	:= TRUE;
            ELSE
                // Second STOP press while hold is active:
                // force a full STOP.
                GVL_HMI.eMachineMode := E_MachineMode.STOPPED;
            END_IF

        // --------------------------------------------------------------------
        // All other modes keep hard STOP behaviour
        // --------------------------------------------------------------------
        ELSE
            GVL_HMI.eMachineMode := E_MachineMode.STOPPED;
    END_CASE

END_IF
END_ACTION

END_PROGRAM

// ---- POUs/2. AutoCycle/PRG_AutoCycle.TcPOU
(*
    PRG_AutoCycle
    -------------------------
    High-level state machine that executes the full automatic cycle of the ASRS:
      - Initialization and safety checks
      - Air supply verification
      - Stage sealing and (optional) metering
      - Leak test
      - Prime solvent lines
      - Recovery, washing and drying phases
      - Post-execution data logging
      - Pause / Hold handling
      - Error handling and safe fallback

    This program is expected to run cyclically while the machine is in AUTO mode
    (e.g. GVL_HMI.eMachineMode = E_MachineMode.AUTO_CYCLE).
*)
PROGRAM PRG_AutoCycle
VAR
    // -----------------------------
    // Global state and basic flags
    // -----------------------------
    CurrentState          : E_MachineStates;     // Current logical state of the auto-cycle state machine
    bErrorFlag            : BOOL;                // Generic error flag (used locally in ERROR_STATE)
    bPowerUpDone          : BOOL := FALSE;       // Indicates that power-up timer has completed at least once
    tonPowerUp            : Tc2_Standard.TON;    // Timer used for initial power-up delay
    bPowerUpTimerComplete : BOOL;                // TRUE when the initial power-up delay has elapsed

    // -----------------------------
    // Initialization stage
    // -----------------------------
    fbInitChecks  : FB_InitChecks;   // FB responsible for initialization safety checks
    bInitCheckDone: BOOL := FALSE;   // TRUE when FB_InitChecks reports initialization OK
    bInitError    : BOOL := FALSE;   // TRUE when FB_InitChecks reports an initialization error

    // -----------------------------
    // Air flow / supply monitoring
    // -----------------------------
    fbAirFlowCheck    : FB_AirFlowCheck; // FB instance that validates main air supply
    bAirSupplyStable  : BOOL;            // TRUE when air supply has been stable above threshold
    bAirSupplyError   : BOOL;            // TRUE if air supply check fails
    rAirSupplyNow     : LREAL;           // Instantaneous air flow / pressure measurement (if needed)

    // -----------------------------
    // Recovery Phase
    // -----------------------------
    fbRecoveryPhase : FB_RecoveryPhase;  // FB that executes the full recovery phase
    aSolenoidSets   : ST_SolenoidSet;    // (Reserved) Solenoid configuration for phases
    bRecoverySuccess: BOOL;              // TRUE when recovery phase completes successfully
    bRecoveryError  : BOOL;              // TRUE when recovery phase fails

    // -----------------------------
    // Washing Phase
    // -----------------------------
    fbWashingPhase  : FB_WashingPhase;   // FB that executes the washing phase
    bWashingSuccess : BOOL;              // TRUE when washing phase completes successfully
    bWashingError   : BOOL;              // TRUE when washing phase fails

    // -----------------------------
    // Drying Phase
    // -----------------------------
    fbDryingPhase  : FB_DryingPhase;     // FB that executes the drying phase
    bDryingSuccess : BOOL;               // TRUE when drying phase completes successfully
    bDryingError   : BOOL;               // TRUE when drying phase fails

    // -----------------------------
    // Seal Stages / Metering
    // -----------------------------
    fbSealStages       : FB_SealStages;       // FB that handles sealing of Andersen stages
    fbMeteringSolvent1 : FB_MeteringSolvent1; // FB for metering solvent 1 during seal if enabled
    bSealStages        : BOOL := FALSE;       // Local execute flag for fbSealStages
    bSealSuccess       : BOOL := FALSE;       // TRUE when sealing operation completes successfully
    bSealError         : BOOL := FALSE;       // TRUE when sealing operation fails

    // -----------------------------
    // Leak Test
    // -----------------------------
    fbLeakTest        : FB_LeakTest;          // FB that performs the leak test routine
    bTestCompleted    : BOOL := FALSE;        // TRUE when the leak test cycle completes
    bTestFailed       : BOOL := FALSE;        // TRUE if the leak test detects a failure
    sTestErrorMessage : STRING := '';         // Leak test error description / details

    // -----------------------------
    // Prime Solvents
    // -----------------------------
    fbPrimeSolvent : FB_PrimeSolvent;         // FB that executes solvent priming routine
    bPrimeDone     : BOOL := FALSE;           // TRUE when priming is completed
    bPrimeError    : BOOL := FALSE;           // TRUE if priming fails

    // -----------------------------
    // Pause / Hold State
    // -----------------------------
    ePauseReturnState   : E_MachineStates;    // State to return to when leaving PAUSE_STATE
    bHoldRequestLatched : BOOL;              // Latched flag for hold request (not fully used here)
    bAnyAxisMoving      : BOOL;              // TRUE if any axis is currently moving (F_AnyAxisMoving)

    // -----------------------------
    // Event / Alarm Triggering
    // -----------------------------
    fbEventHandler : FB_EventHandler;        // Generic event/alarm logger
    bExecuteEvent  : BOOL := FALSE;          // Rising edge triggers event execution
    bEventDone     : BOOL := FALSE;          // TRUE when event handling is finished
    sSystem        : STRING(256);            // System / subsystem identifier for event log
    sMessage       : STRING(256);            // Human-readable event description
	
	// -----------------------------
    // Database Interaction
    // -----------------------------
	bDBPostRunInsert : BOOL := FALSE;		//Insert Command sent flag 

	
END_VAR

// ==========================================================================
// 1) Detect if any axis is still moving
//    This is used by the HOLD / PAUSE logic to avoid interrupting moves
//    mid-motion. The state machine only enters PAUSE_STATE when all
//    axes are stopped, so we pause between movements, not in the middle.
// ==========================================================================
bAnyAxisMoving := F_AnyAxisMoving();

// ==========================================================================
// 2) HOLD request handling (global "Pause" behavior)
//
//    If the operator requests a HOLD (bAutoCycleHoldReq = TRUE) while:
//      - the machine is running auto cycle,
//      - no other hold is already active,
//      - and no axis is currently moving,
//    then:
//      - Capture the current state as the "return state"
//      - Mark HOLD as active
//      - Open the HOLD popup on the HMI
//      - Jump to PAUSE_STATE
//
//    This allows pausing between macro-steps without losing the current
//    state machine context.
// ==========================================================================
IF GVL_HMI.bAutoCycleHoldReq
   AND NOT GVL_HMI.bAutoCycleHoldActive
   AND NOT bAnyAxisMoving
THEN
    // We are pausing between "macro-steps", so the return state
    // is the current state of the auto-cycle.
    ePauseReturnState            := CurrentState;

    // Mark hold as active and consume the request
    GVL_HMI.bAutoCycleHoldActive := TRUE;
    GVL_HMI.bAutoCycleHoldReq    := FALSE;

    // Open the HOLD popup on HMI
    GVL_HMI.bAutoCycleHoldPopup  := TRUE;

    // Enter PAUSE_STATE. Execution below is skipped this cycle.
    CurrentState := E_MachineStates.PAUSE_STATE;
    RETURN;
END_IF

// ==========================================================================
// 3) Auto Cycle State Machine
// ==========================================================================
CASE CurrentState OF

    // ----------------------------------------------------------------------
    // INIT
    //  - Check power supplies, doors and air supply interlocks.
    //  - Only proceeds to air flow check when all conditions are OK.
    //  - Any error drives the machine to ERROR_STATE.
    // ----------------------------------------------------------------------
    E_MachineStates.INIT:

        // Log info event: Initialization is being checked
        sSystem  := 'StateMachine.INIT';
        sMessage := 'Cheking Safety Conditions!'; // NOTE: text used as-is to keep compatibility
        fbEventHandler(
            bExecute   := bExecuteEvent,
            eEventName := E_Events.INFO,
            sSystem    := sSystem,
            sMessage   := sMessage,
            bDone      => bEventDone
        );
        ResetEventTrigger();

        // Execute FB responsible for all initial operation checks
        fbInitChecks(
            bPower24V_OK := GVL_IO.gDigInputs.b24VPowerSupplyOK,
            bPower48V_OK := GVL_IO.gDigInputs.b48VPowerSupplyOK,
            bDoorsClosed := GVL_Safety.bDoorClosedAlias,
            bDoorsLocked := GVL_Safety.bDoorLockedFeedback,
            // Air supply currently re-used from door "below" feedback
            bAirEnabled  := GVL_Safety.SafetyOutputs.bBelowDoorsFeedback,
            bExecute     := TRUE,
            bReset       := FALSE,
            bInitOK      => bInitCheckDone,
            bError       => bInitError
        );

        // --- State transitions based on initialization result ---
        IF bInitError THEN
            // Log error and go to ERROR_STATE
            sSystem  := 'StateMachine.INIT';
            sMessage := 'Initialization fail - Going to Error State!';
            fbEventHandler(
                bExecute   := bExecuteEvent,
                eEventName := E_Events.ERROR,
                sSystem    := sSystem,
                sMessage   := sMessage,
                bDone      => bEventDone
            );
            ResetEventTrigger();

            CurrentState := E_MachineStates.ERROR_STATE;

        ELSIF bInitCheckDone THEN
            // Initialization successful: log and start post-run tracking
            sSystem  := 'StateMachine.INIT';
            sMessage := 'Initialization Successful!';
            fbEventHandler(
                bExecute   := bExecuteEvent,
                eEventName := E_Events.INFO,
                sSystem    := sSystem,
                sMessage   := sMessage,
                bDone      => bEventDone
            );
            ResetEventTrigger();

            // Start post-run info record (start time and DB select)
            GVL_DB.stPostRunInfo.timeEventStarted := TO_STRING(TIME());
            DB_Query.state := E_DB_QUERY_STATE.SELECT_POST_LAST_RUN;

            // Proceed to air flow check
            CurrentState := E_MachineStates.CHECK_AIR_FLOW;
        END_IF;


    // ----------------------------------------------------------------------
    // CHECK_AIR_FLOW
    //  - Validates that main air supply is above configured threshold
    //    and remains stable for a given time.
    //  - Any sensor or stability error sends the machine to ERROR_STATE.
    // ----------------------------------------------------------------------
    E_MachineStates.CHECK_AIR_FLOW:

        // 1. Check if the pressure sensor reports an error state
        IF GVL_IO.gAnalogInputs.bPressureRegulatorError THEN
            // Log sensor error
            fbEventHandler(
                bExecute   := bExecuteEvent,
                eEventName := E_Events.ERROR,
                sSystem    := 'Air Supply Check',
                sMessage   := 'Air Supply Sensor Error State!',
                bDone      => bEventDone
            );
            ResetEventTrigger();

            // Go to ERROR_STATE and mark local error flag
            CurrentState    := E_MachineStates.ERROR_STATE;
            bAirSupplyError := TRUE;
        ELSE
            // 2. Execute airflow verification (threshold + stabilization time)
            fbAirFlowCheck(
                iRawSensorValue    := GVL_IO.gAnalogInputs.rMainPressureSupplyInput,  // Raw sensor input
                iSensorID          := 1,                                              // FESTO air supply sensor ID
                rPressureThreshold := GVL_Settings.rAirSupplyThreshold,               // Minimum pressure
                tStabilizationTime := GVL_Settings.rAirSupplyTestingTime,             // Time to remain stable
                bExecute           := TRUE,
                bReset             := FALSE,
                bAirFlowOK         => bAirSupplyStable,
                bAirFlowError      => bAirSupplyError
            );

            // 3. State transitions based on air flow result
            IF bAirSupplyError THEN
                // Any error drives to ERROR_STATE and activates tower red light
                CurrentState := E_MachineStates.ERROR_STATE;
                GVL_IO.gDigOutputs.bTowerRedLight := TRUE;

            ELSIF bAirSupplyStable THEN
                // Air supply OK → proceed to sealing stages
                CurrentState := E_MachineStates.SEAL_STAGES;
            END_IF;
        END_IF;


    // ----------------------------------------------------------------------
    // SEAL_STAGES
    //  - Close and seal Andersen stages.
    //  - Optionally execute metering of solvent 1 in parallel (if enabled).
    //  - On success → LEAK_TEST, on any error → ERROR_STATE.
    // ----------------------------------------------------------------------
    E_MachineStates.SEAL_STAGES:

        // Enable sealing logic only if M1 STO is enabled (safety condition)
        IF GVL_Safety.bM1STOEnabled THEN
            bSealStages := TRUE;
        ELSE
            bSealStages := FALSE;
        END_IF

        // Execute sealing stages FB
        fbSealStages(bExecute := bSealStages);

        // Optional metering of solvent 1 during seal step
        IF GVL_Settings.bGeneralSealAndPump THEN
            fbMeteringSolvent1(bExecute := TRUE);
        END_IF

        // Error check for both sealing and metering
        IF fbSealStages.bSealError OR fbMeteringSolvent1.bError THEN
            CurrentState := E_MachineStates.ERROR_STATE;
        END_IF

        // State transitions on success
        IF NOT GVL_Settings.bGeneralSealAndPump THEN
            // Only sealing required
            IF fbSealStages.bSealSuccess AND NOT fbSealStages.bSealError THEN
                CurrentState := E_MachineStates.LEAK_TEST;
            END_IF
        ELSE
            // Seal + metering required
            IF fbSealStages.bSealSuccess
               AND fbMeteringSolvent1.bDone
               AND NOT fbSealStages.bSealError
               AND NOT fbMeteringSolvent1.bError
            THEN
                // Mark metering complete and reset FB before proceeding
                GVL_Settings.bMeteringSolvent1Done := TRUE;

                IF fbMeteringSolvent1.Reset() THEN
                    CurrentState := E_MachineStates.LEAK_TEST;
                END_IF
            END_IF
        END_IF


    // ----------------------------------------------------------------------
    // LEAK_TEST
    //  - Performs leak test using FB_LeakTest with configured timing.
    //  - On success → PRIME_SOLVENT, on failure → ERROR_STATE.
    // ----------------------------------------------------------------------
    E_MachineStates.LEAK_TEST:

        // Call the Leak Test function block
        fbLeakTest(
            bExecute          := TRUE,
            eSolenoidPosition := E_SolenoidSet.LEAKTEST, // Configure solenoids for leak test
            tMonitorTime      := GVL_Settings.stLeakTestParameters.tLeakTestMonitorTime,
            tPressureUpTime   := GVL_Settings.stLeakTestParameters.tLeakTestBuildUpTime,
            bLeakTestDone     => bTestCompleted,
            bLeakTestError    => bTestFailed,
            sLTMessageError   => sTestErrorMessage
        );

        // Transitions based on leak test result
        IF bTestCompleted THEN
			// Return solenoids to idle / safe position
        	GVL_IO.gSetSolenoidControl.Idle();
            // Leak test OK → proceed to priming
            CurrentState := E_MachineStates.PRIME_SOLVENT;

        ELSIF bTestFailed THEN
			// Return solenoids to idle / safe position
        	GVL_IO.gSetSolenoidControl.Idle();
            // Leak test failed → go to ERROR_STATE
            CurrentState := E_MachineStates.ERROR_STATE;
        END_IF;


    // ----------------------------------------------------------------------
    // PRIME_SOLVENT
    //  - Primes all necessary solvent lines according to recipe/settings.
    //  - On success → RECOVERY_PHASE, on error → ERROR_STATE.
    // ----------------------------------------------------------------------
    E_MachineStates.PRIME_SOLVENT:
	
	IF GVL_HMI.bAutoCyclePrimeSolvents THEN
		// Execute PrimeSolvent FB
        fbPrimeSolvent(bExecute := TRUE);

        // Capture FB outputs for clarity
        bPrimeDone  := fbPrimeSolvent.bDone;
        bPrimeError := fbPrimeSolvent.bError;

        // Evaluate prime result
        IF bPrimeError THEN
            CurrentState := E_MachineStates.ERROR_STATE;

        ELSIF bPrimeDone THEN
            // Optionally reset FB instance before moving on
            IF fbPrimeSolvent.Reset() THEN
                CurrentState := E_MachineStates.RECOVERY_PHASE;
            END_IF
        END_IF
	ELSE
		GVL_HMI.HMIAnimation.sLoadTextPrime  := 'Prime Skipped';
        GVL_HMI.HMIAnimation.rLoadBarPrime   := 100.0;
        GVL_HMI.HMIAnimation.eIconStatePrime := E_IconState.Completed;
		CurrentState := E_MachineStates.RECOVERY_PHASE;
	END_IF

        


    // ----------------------------------------------------------------------
    // RECOVERY_PHASE
    //  - Executes the full recovery of particles/solvents from stages.
    //  - On success → WASHING_PHASE, on error → ERROR_STATE.
    // ----------------------------------------------------------------------
    E_MachineStates.RECOVERY_PHASE:

        // Execute Recovery Phase FB
        fbRecoveryPhase(bExecute := TRUE);

        // Capture result flags
        bRecoverySuccess := fbRecoveryPhase.bSuccess;
        bRecoveryError   := fbRecoveryPhase.bError;

        // State transitions based on FB result
        IF bRecoveryError THEN
            CurrentState := E_MachineStates.ERROR_STATE;
        ELSIF bRecoverySuccess THEN
            CurrentState := E_MachineStates.WASHING_PHASE;
        END_IF;


    // ----------------------------------------------------------------------
    // WASHING_PHASE
    //  - Executes the washing routine after recovery.
    //  - On success → DRYING_PHASE, on error → ERROR_STATE.
    // ----------------------------------------------------------------------
    E_MachineStates.WASHING_PHASE:

        // Execute Washing Phase FB
        fbWashingPhase(bExecute := TRUE);

        // Capture result flags
        bWashingSuccess := fbWashingPhase.bWashingDone;
        bWashingError   := fbWashingPhase.bWashingError;

        // State transitions based on FB result
        IF bWashingError THEN
            CurrentState := E_MachineStates.ERROR_STATE;
        ELSIF bWashingSuccess THEN
            CurrentState := E_MachineStates.DRYING_PHASE;
        END_IF;


    // ----------------------------------------------------------------------
    // DRYING_PHASE
    //  - Executes the drying routine after washing.
    //  - On success → POST_EXECUTION, on error → ERROR_STATE.
    // ----------------------------------------------------------------------
    E_MachineStates.DRYING_PHASE:

        // Execute Drying Phase FB
        fbDryingPhase(bExecute := TRUE);

        // Capture result flags
        bDryingSuccess := fbDryingPhase.bDryingDone;
        bDryingError   := fbDryingPhase.bDryingError;

        // State transitions based on FB result
        IF bDryingError THEN
            CurrentState := E_MachineStates.ERROR_STATE;
        ELSIF bDryingSuccess THEN
            CurrentState := E_MachineStates.POST_EXECUTION;
        END_IF;


    // ----------------------------------------------------------------------
    // POST_EXECUTION
    //  - Collects and stores post-run information for reporting.
    //  - Triggers DB insert and returns machine to STOPPED mode.
    // ----------------------------------------------------------------------
    E_MachineStates.POST_EXECUTION:

        // Fill post-run info structure with timing and recipe data
        GVL_DB.stPostRunInfo.timeEventCompleted  := TO_STRING(TIME());
        GVL_DB.stPostRunInfo.runNo              := GVL_DB.stPostRunReport[0].runNo + 1;
        GVL_DB.stPostRunInfo.comment            := GVL_HMI.sAutoCycleComment;
        GVL_DB.stPostRunInfo.analyst            := '';
        GVL_DB.stPostRunInfo.CalibrationNo      := 0;
        GVL_DB.stPostRunInfo.emptyTubesFactor   := TO_STRING(GVL_Settings.stPumpParameters.iEmptyFactor);
        GVL_DB.stPostRunInfo.fillTubesFactor    := TO_STRING(GVL_Settings.stPumpParameters.iFillolventTubesFactor);
        GVL_DB.stPostRunInfo.meterVelocity      := TO_STRING(GVL_Settings.stPumpParameters.iMeterVelocity);
        GVL_DB.stPostRunInfo.methodID           := GVL_HMI.stRecipeInfo.iRevision;
        GVL_DB.stPostRunInfo.runVelocity        := TO_STRING(GVL_Settings.stPumpParameters.iRunVelocity);
        GVL_DB.stPostRunInfo.softwareVersion    := '';
        GVL_DB.stPostRunInfo.solvent1NameRevision := '';
        GVL_DB.stPostRunInfo.solvent2NameRevision := '';
        GVL_DB.stPostRunInfo.solvent3NameRevision := '';
        GVL_DB.stPostRunInfo.solvent4NameRevision := '';
        GVL_DB.stPostRunInfo.sysMasterRevision    := '';
        GVL_DB.stPostRunInfo.sysSettingsRevision  := '';

  		// Database post run insert 
		IF NOT DB_Query.bBusyDb THEN
			// Request DB insert of the new run record
        	DB_Query.state := E_DB_QUERY_STATE.INSERT_RUN;
			bDBPostRunInsert := TRUE;
		ELSIF NOT DB_Query.bBusyDb AND bDBPostRunInsert THEN
			// When finished, hand control back to STOPPED mode
        	GVL_HMI.eMachineMode := E_MachineMode.STOPPED;
			bDBPostRunInsert := FALSE;
		END_IF
        
    // ----------------------------------------------------------------------
    // PAUSE_STATE
    //  - Neutral wait state when the auto-cycle is on HOLD.
    //  - The operator can:
    //      - CONTINUE: resume exactly from ePauseReturnState
    //      - CANCEL: abort the run and go to STOPPED / SystemInit
    // ----------------------------------------------------------------------
    E_MachineStates.PAUSE_STATE:

        // Ensure popup remains active while in pause
        GVL_HMI.bAutoCycleHoldPopup := TRUE;

        // CONTINUE: resume from the previously stored state
        IF GVL_HMI.bAutoCycleContinueCmd THEN

            GVL_HMI.bAutoCycleContinueCmd := FALSE;
            GVL_HMI.bAutoCycleHoldActive  := FALSE;
            GVL_HMI.bAutoCycleHoldPopup   := FALSE;
            // Note: we do not re-assert bAutoCycleHoldReq here

            // Resume at the same logical state where the pause occurred
            CurrentState := ePauseReturnState;
            // The FBs in that state will see that no moves are in progress
            // and will continue with the next sub-step in their internal logic.

        // CANCEL: abort current run and go back to STOPPED State
        ELSIF GVL_HMI.bAutoCycleCancelCmd THEN

            GVL_HMI.bAutoCycleCancelCmd  := FALSE;
            GVL_HMI.bAutoCycleHoldActive := FALSE;
            GVL_HMI.bAutoCycleHoldPopup  := FALSE;
            GVL_HMI.bAutoCycleHoldReq    := FALSE;

            // Switch machine mode to STOPPED. PRG_StoppedState will take over.
            GVL_HMI.eMachineMode := E_MachineMode.STOPPED;

        END_IF


    // ----------------------------------------------------------------------
    // ERROR_STATE
    //  - Generic error handling state for the auto-cycle.
    //  - Ensures safe outputs (e.g. tower red light, solenoids idle).
    //  - Machine remains in STOPPED mode until reset logic is applied.
    // ----------------------------------------------------------------------
    E_MachineStates.ERROR_STATE:

        // Signal error via tower light
        GVL_IO.gDigOutputs.bTowerRedLight := TRUE;

        // Return solenoids to idle / safe position
        GVL_IO.gSetSolenoidControl.Idle();

        // Force machine mode to STOPPED; PRG_StoppedState will manage reset
        GVL_HMI.eMachineMode := E_MachineMode.STOPPED;

        // Simple example of local error reset logic:
        // if the physical stop button is pressed, clear the local flag
        // and send the state machine back to INIT.
        IF GVL_IO.gDigInputs.bStopButton THEN
            bErrorFlag   := FALSE;
            CurrentState := E_MachineStates.INIT;
        END_IF;

END_CASE;

METHOD Reset : BOOL
VAR_INPUT
END_VAR
// Reset FBs and flags
fbInitChecks(bExecute := FALSE, bReset := TRUE);
fbAirFlowCheck(bExecute := FALSE, bReset := TRUE);
fbSealStages(bExecute := FALSE);
fbLeakTest(bExecute := FALSE);
fbRecoveryPhase(bExecute := FALSE);
fbEventHandler(bExecute := FALSE);

//Resets the state machine
CurrentState := E_MachineStates.INIT;

//Reset the HMI Icons animation
GVL_HMI.HMIAnimation.eIconStateAirFlow 	:= E_IconState.Waiting;
GVL_HMI.HMIAnimation.eIconStateSealing	:= E_IconState.Waiting;
GVL_HMI.HMIAnimation.eIconStateHardware := E_IconState.Waiting;
GVL_HMI.HMIAnimation.eIconStatePrime 	:= E_IconState.Waiting;
GVL_HMI.HMIAnimation.eIconStateLeakTest := E_IconState.Waiting;
GVL_HMI.HMIAnimation.eIconStateRecovery := E_IconState.Waiting;
GVL_HMI.HMIAnimation.eIconStateWashing 	:= E_IconState.Waiting;
GVL_HMI.HMIAnimation.eIconStateDry 		:= E_IconState.Waiting;

// Reset State flags
bInitCheckDone 		:= FALSE;
bInitError 			:= FALSE;
bAirSupplyStable 	:= FALSE;
bAirSupplyError 	:= FALSE;
bSealSuccess 		:= FALSE;
bSealError 			:= FALSE;
bTestCompleted 		:= FALSE;
bTestFailed 		:= FALSE;
sTestErrorMessage 	:= '';
bRecoverySuccess 	:= FALSE;
bRecoveryError 		:= FALSE;
bErrorFlag 			:= FALSE;
bExecuteEvent 		:= FALSE;
bEventDone 			:= FALSE;
bDBPostRunInsert 	:= FALSE;

// Auto Cycle FB's Reset	
IF  fbSealStages.Reset() 
    AND fbRecoveryPhase.Reset() 
    AND fbLeakTest.Reset() 
    AND fbMeteringSolvent1.Reset() 
    AND fbAirFlowCheck.Reset() 
    AND fbInitChecks.Reset()
    AND fbWashingPhase.Reset()
    AND fbDryingPhase.Reset()
    AND fbPrimeSolvent.Reset() THEN  
		Reset := TRUE;
		RETURN;
ELSE
	Reset := FALSE;
END_IF
END_METHOD

ACTION ResetEventTrigger:
IF bEventDone THEN
        bExecuteEvent := FALSE;
        bEventDone := FALSE;
END_IF;
END_ACTION

END_PROGRAM

// ---- POUs/2. AutoCycle/Stages/FB_InitChecks.TcPOU
(*
==============================================================================
 FB_InitChecks
------------------------------------------------------------------------------
 Purpose:
   Perform the machine initialization safety validation before starting 
   Auto Cycle or any motion-critical operation.

   This block verifies the following conditions in sequence:
     1) 24V and 48V power supply availability  
     2) All safety doors are physically closed  
     3) Doors are locked (interlock engaged)  
     4) Air supply is available and safe to enable  
     5) If all checks pass → bInitOK := TRUE

 Usage:
   - Call cyclically.
   - Set bExecute := TRUE to start evaluation.
   - bInitOK  = TRUE  → All initial conditions satisfied.
   - bError   = TRUE  → A condition failed; machine must not start.
   - bReset   = TRUE  → Asynchronous reset to return FB to state 0.

 Safety Outputs Controlled:
   - GVL_Safety.bAirSupplyEnable   : Enables solenoid / pneumatic air supply.
   - GVL_Safety.bDoorLockCommand   : Locks the safety doors.
   - GVL_Safety.SafetyOutputs.bAirPressureOK : Temporary mock (TODO).

 Notes:
   - State machine steps:
       0 : Reset / Idle  
       1 : Check power  
       2 : Check doors closed  
       3 : Check doors locked  
       4 : Enable air supply  
       5 : Success  
      99 : Error state  
==============================================================================
*)
FUNCTION_BLOCK FB_InitChecks
VAR_INPUT
    bExecute      : BOOL;   // Start initialization check
    bPower24V_OK  : BOOL;   // External 24V supply OK
    bPower48V_OK  : BOOL;   // External 48V supply OK
    bDoorsClosed  : BOOL;   // Physical door closed sensors
    bDoorsLocked  : BOOL;   // Door lock feedback
    bAirEnabled   : BOOL;   // Air supply feedback (valves/sensors)
    bReset        : BOOL;   // Asynchronous reset
END_VAR

VAR_OUTPUT
    bInitOK : BOOL := FALSE; // TRUE when all safety checks pass
    bError  : BOOL := FALSE; // TRUE if any condition fails
END_VAR

VAR
    iState : INT := 0;       // Internal state machine
END_VAR

// ==========================================================================
// Initialization State Machine
// ==========================================================================
CASE iState OF

    // ----------------------------------------------------------------------
    // STATE 0 — RESET / IDLE
    // ----------------------------------------------------------------------
    0:
        // Reset outputs
        bInitOK := FALSE;
        bError  := FALSE;

        // Reset safety commands
        GVL_Safety.bAirSupplyEnable := FALSE;
        GVL_Safety.bDoorLockCommand := FALSE;

        // Start sequence
        IF bExecute AND NOT bReset THEN
            iState := 1;   // Next: power supply check
        END_IF


    // ----------------------------------------------------------------------
    // STATE 1 — POWER SUPPLY CHECK
    // ----------------------------------------------------------------------
    1:
        IF bReset THEN
            iState := 0;   // Full reset if requested

        ELSIF NOT (bPower24V_OK AND bPower48V_OK) THEN
            // Fail: power missing
            bError := TRUE;

            GVL_Safety.bAirSupplyEnable := FALSE;
            GVL_Safety.bDoorLockCommand := FALSE;

            iState := 99;  // Error state

        ELSE
            iState := 2;   // Pass → next check
        END_IF;


    // ----------------------------------------------------------------------
    // STATE 2 — DOORS CLOSED CHECK
    // ----------------------------------------------------------------------
    2:
        IF bReset THEN
            iState := 0;

        ELSIF NOT bDoorsClosed THEN
            // Fail: a door is open
            GVL_Safety.bAirSupplyEnable := FALSE;
            GVL_Safety.bDoorLockCommand := FALSE;

            iState := 99;

        ELSE
            iState := 3;   // Pass → next
        END_IF;


    // ----------------------------------------------------------------------
    // STATE 3 — DOOR LOCK CHECK
    // ----------------------------------------------------------------------
    3:
        IF bReset THEN
            iState := 0;

        ELSIF NOT bDoorsLocked THEN
            (* NOTE:
               In the original system, the door locking command might be issued here.
               For now, it is commented out due to testing state of the machine.
               TODO: Restore door locking command when hardware is validated:
                 GVL_Safety.bDoorLockCommand := TRUE;
            *)
            GVL_Safety.bAirSupplyEnable := FALSE;

        ELSE
            iState := 4;   // Pass → proceed to air supply
        END_IF;


    // ----------------------------------------------------------------------
    // STATE 4 — AIR SUPPLY CHECK
    // ----------------------------------------------------------------------
    4:
        IF bReset THEN
            iState := 0;

        ELSIF NOT bAirEnabled THEN
            // Temporary: assert air pressure OK (mock)
            // TODO: Replace with actual analog pressure measurement
            GVL_Safety.SafetyOutputs.bAirPressureOK := TRUE;

            GVL_Safety.bAirSupplyEnable := TRUE;

        ELSE
            // Air OK → move to final state
            iState := 5;
        END_IF;


    // ----------------------------------------------------------------------
    // STATE 5 — SUCCESS (ALL CHECKS PASSED)
    // ----------------------------------------------------------------------
    5:
        IF bReset THEN
            iState := 0;
        ELSE
            bInitOK := TRUE;
        END_IF;


    // ----------------------------------------------------------------------
    // STATE 99 — ERROR STATE
    // ----------------------------------------------------------------------
    99:
        IF bReset THEN
            iState := 0;
        ELSE
            bError := TRUE;
        END_IF;

END_CASE

(*
==============================================================================
 Method: Reset
------------------------------------------------------------------------------
 Purpose:
   Restore internal state to default so a new initialization sequence 
   may be executed safely.

 Behaviour:
   - Clears bInitOK, bError.
   - Returns to state 0.
   - Does NOT automatically re-enable safety outputs (left to state machine).
==============================================================================
*)
METHOD Reset : BOOL
VAR_INPUT
END_VAR
Reset := FALSE;

// Clear flags
bInitOK := FALSE;
bError  := FALSE;

// Reset internal FSM
iState := 0;

// Method completes successfully
Reset := TRUE;
RETURN;
END_METHOD

END_FUNCTION_BLOCK

// ---- POUs/2. AutoCycle/Stages/FB_AirFlowCheck.TcPOU
(*
==============================================================================
 FB_AirFlowCheck
------------------------------------------------------------------------------
 Purpose:
   - Validate that the main air supply / airflow is above a minimum threshold
     and remains stable for a configured stabilization time.

 Behaviour:
   - Inputs:
       iRawSensorValue   : Raw value from analog pressure sensor (16-bit).
       iSensorID         : Which sensor type is in use (1 = Festo, 2 = SMC).
       rPressureThreshold: Minimum acceptable pressure for "OK" condition.
       tStabilizationTime: Time that pressure must stay above threshold.
       bExecute          : Command to start the check.
       bReset            : Asynchronous reset for this FB.

   - Outputs:
       bAirFlowOK        : TRUE when pressure ≥ threshold for the whole
                           stabilization time.
       bAirFlowError     : TRUE when pressure < threshold, or check fails.

   - Internal steps (iState):
       0: Reset / Idle
       1: Read and scale sensor
       2: Compare pressure against threshold
       3: Wait for stabilization timer to elapse
       4: Completed successfully
      99: Error state

   - HMI:
       - Action ACT_HMIProgressBar updates:
           GVL_HMI.HMIAnimation.sLoadTextAirFlow
           GVL_HMI.HMIAnimation.rLoadBarAirFlow
           GVL_HMI.HMIAnimation.eIconStateAirFlow

 Usage:
   - Call cyclically.
   - Set bExecute := TRUE to start the airflow verification.
   - Check bAirFlowOK / bAirFlowError.
   - Use method Reset() to bring FB back to a clean state if needed.
==============================================================================
*)
FUNCTION_BLOCK FB_AirFlowCheck
VAR_INPUT
    iRawSensorValue    : INT;   // Raw sensor value (16-bit)
    iSensorID          : INT;   // Sensor ID (1 = Festo, 2 = SMC)
    rPressureThreshold : REAL;  // Minimum air pressure threshold
    tStabilizationTime : TIME;  // Required stabilization time above threshold
    bExecute           : BOOL;  // Signal to start verification
    bReset             : BOOL;  // Reset command
END_VAR

VAR_OUTPUT
    bAirFlowOK    : BOOL;       // TRUE if airflow is within acceptable limits
    bAirFlowError : BOOL;       // TRUE if airflow check failed
END_VAR

VAR
    iState               : INT := 0;          // State machine variable
    TON_Stabilization    : TON;              // Stabilization timer
    fbSensorScaling      : FB_SensorScaling; // Sensor scaling function block
    rConvertedPressure   : REAL;             // Scaled pressure value
    bTimerActive         : BOOL;             // Internal flag to keep the timer running
    bProgressBarComplete : BOOL := FALSE;    // HMI progress bar completion latch
END_VAR

// -----------------------------------------------------------------------------
// HMI Progress Bar Animation for Air Flow / Init Sequence
// -----------------------------------------------------------------------------
ACT_HMIProgressBar();

// -----------------------------------------------------------------------------
// Air Flow Check State Machine
// -----------------------------------------------------------------------------
CASE iState OF

    //=====================================================================
    // 0) RESET / IDLE
    //    - Clear outputs and internal flags.
    //    - Wait for bExecute to start verification (if not resetting).
    //=====================================================================
    0:
        bAirFlowOK          := FALSE;
        bAirFlowError       := FALSE;
        TON_Stabilization(IN := FALSE);
        rConvertedPressure  := 0.0;
        bTimerActive        := FALSE;

        IF bExecute AND NOT bReset THEN
            iState := 1;  // Proceed to airflow verification
        END_IF


    //=====================================================================
    // 1) START VERIFICATION
    //    - Optionally handle reset.
    //    - Trigger sensor scaling (raw → engineering units).
    //=====================================================================
    1:
        IF bReset THEN
            iState := 0;  // Go back to reset state if requested

        ELSIF bExecute THEN
            // Convert the raw sensor value before checking airflow
            fbSensorScaling(
                iRawValue := iRawSensorValue,
                iSensorID := iSensorID,
                rPressure => rConvertedPressure
            );

            iState := 2;  // Proceed to pressure check
        END_IF;


    //=====================================================================
    // 2) PRESSURE CHECK
    //    - Compare scaled pressure against threshold.
    //      * If ≥ threshold → start stabilization timer.
    //      * If < threshold → set error and go to error state.
    //=====================================================================
    2:
        IF bReset THEN
            iState := 0;  // Ensure reset if requested

        ELSIF rConvertedPressure >= rPressureThreshold THEN
            // Pressure is high enough, start stabilization timing
            bTimerActive := TRUE;
            TON_Stabilization(IN := bTimerActive, PT := tStabilizationTime);

            iState := 3;  // Proceed to stabilization time check
        ELSE
            // Pressure below threshold → immediate error
            bTimerActive := FALSE;
            TON_Stabilization(IN := FALSE);

            bAirFlowOK   := FALSE;
            bAirFlowError:= TRUE;

            iState := 99; // Move to error state
        END_IF;


    //=====================================================================
    // 3) STABILIZATION TIME
    //    - Require pressure to stay ≥ threshold for the entire
    //      tStabilizationTime.
    //=====================================================================
    3:
        IF bReset THEN
            iState := 0;  // Ensure reset if requested

        ELSIF TON_Stabilization.Q THEN
            // Stabilization time elapsed with acceptable pressure
            bTimerActive := FALSE;
            TON_Stabilization(IN := FALSE);  // Stop the timer

            iState := 4;  // Proceed to final state
        ELSE
            // Keep timer running while we are waiting
            TON_Stabilization(IN := bTimerActive, PT := tStabilizationTime);
        END_IF;


    //=====================================================================
    // 4) COMPLETED
    //    - Airflow successfully verified.
    //=====================================================================
    4:
        IF bReset THEN
            iState := 0;  // Allow clean reset from final state
        END_IF;

        // Prepare progress bar for next cycle and set outputs
        bProgressBarComplete := FALSE;
        bAirFlowOK           := TRUE;
        bAirFlowError        := FALSE;


    //=====================================================================
    // 99) ERROR STATE
    //    - Airflow check failed (pressure below threshold).
    //=====================================================================
    99:
        IF bReset THEN
            iState := 0;  // Ensure reset from error state
        ELSE
            bAirFlowError := TRUE;
        END_IF;

END_CASE

ACTION ACT_HMIProgressBar:
(*
==============================================================================
 ACT_HMIProgressBar
------------------------------------------------------------------------------
 Purpose:
   - Provide a simple, state-based progress indication (0–100%) for the
     airflow / init check in the HMI.
   - Maps internal state iState to a fixed bar percentage and updates:
        GVL_HMI.HMIAnimation.sLoadTextAirFlow
        GVL_HMI.HMIAnimation.rLoadBarAirFlow
        GVL_HMI.HMIAnimation.eIconStateAirFlow

 Notes:
   - This is a coarse progress indicator; it does not use real timing.
==============================================================================
*)

// Static text and default icon while the check is in progress
IF NOT bProgressBarComplete THEN
    GVL_HMI.HMIAnimation.sLoadTextAirFlow  := 'Init Checks';
    GVL_HMI.HMIAnimation.rLoadBarAirFlow   := 0.0;
    GVL_HMI.HMIAnimation.eIconStateAirFlow := E_IconState.InProgress;
END_IF

// Map state machine to a simple 0–100% progress value
CASE iState OF
    0:  // State 0: Idle / reset
        GVL_HMI.HMIAnimation.rLoadBarAirFlow := 0.0;

    1:  // State 1: Start verification
        GVL_HMI.HMIAnimation.rLoadBarAirFlow := 25.0;

    2:  // State 2: Threshold comparison
        GVL_HMI.HMIAnimation.rLoadBarAirFlow := 50.0;

    3:  // State 3: Stabilization time
        GVL_HMI.HMIAnimation.rLoadBarAirFlow := 75.0;

    4:  // State 4: Airflow verification completed
        GVL_HMI.HMIAnimation.rLoadBarAirFlow := 100.0;

        // Mark icon as completed when initialization is OK
        GVL_HMI.HMIAnimation.eIconStateAirFlow := E_IconState.Completed;
        bProgressBarComplete := TRUE;

    99: // State 99: Error state
        GVL_HMI.HMIAnimation.rLoadBarAirFlow := 0.0;
END_CASE
END_ACTION

(*
==============================================================================
 Method: Reset
------------------------------------------------------------------------------
 Purpose:
   - Reset FB_AirFlowCheck to a known idle state so that a new airflow check
     can start cleanly.

 Behaviour:
   - Clears:
       * Outputs: bAirFlowOK, bAirFlowError
       * State machine: iState
       * Internal flags: bTimerActive, bProgressBarComplete
       * Internal values: rConvertedPressure
       * Timer TON_Stabilization
       * HMI icon state for AirFlow

   - Returns:
       Reset = TRUE  (always, after executing reset logic)
==============================================================================
*)
METHOD Reset : BOOL
VAR_INPUT
END_VAR
Reset := FALSE;

// Clear public outputs
bAirFlowOK    := FALSE;
bAirFlowError := FALSE;

// Reset internal state machine and values
iState               := 0;
rConvertedPressure   := 0.0;
bTimerActive         := FALSE;
bProgressBarComplete := FALSE;

// Stop and reset stabilization timer
TON_Stabilization(IN := FALSE);

// Reset HMI icon to "Waiting" state
GVL_HMI.HMIAnimation.eIconStateAirFlow := E_IconState.Waiting;

// Indicate reset completed
Reset := TRUE;
RETURN;
END_METHOD

END_FUNCTION_BLOCK

// ---- POUs/Utilities/FB_SensorScaling.TcPOU
FUNCTION_BLOCK FB_SensorScaling
VAR_INPUT
	iRawValue 	: INT;  //EL3058 raw meassure 16bits
	iSensorID	: INT;	//Sensor ID [1 for Festo | 2 for SMC Pressure Regulator | 3 for SMC PSE550-28 Leak Test sensor]
END_VAR
VAR_OUTPUT
	rPressure 	: REAL; //Pressure output in Bar
END_VAR
VAR
	rScalingFactor : REAL;
    rOffset        : REAL;
END_VAR

// Scaling definition for each sensor
CASE iSensorID OF
    1:  // Festo MS6: 4-20mA | 0-6 bar
        rScalingFactor := 0.0003156;
        rOffset := -0.115;
		
    2:  // SMC ISE/ZSE20: 4-20mA | -0.100 to 1.000 MPa [1.0 to 10.0 bar]
        rScalingFactor := 11.0 / (16384 - 3277); // 11 Bar Range
        rOffset := -1.0;  // Starts at -1.0 Bar
		
	3: // SMC PSE550-28: 4-20mA | -50 to 50kPa [-0.5 to 0.5 bar]
        rScalingFactor := 0.0002442;  // 1 bar range over 4095 steps
        rOffset := -0.5; // Starts at -0.5 bar
		
    ELSE
        rScalingFactor := 1.0;
        rOffset := 0.0;
END_CASE

// Applying the scaling
rPressure := rScalingFactor * TO_REAL(iRawValue) + rOffset;

END_FUNCTION_BLOCK

// ---- POUs/2. AutoCycle/Stages/FB_RecoveryPhase.TcPOU
(*
    FB_RecoveryPhase
    ------------------------------------------------------------------------
    Purpose:
      - Orchestrates the full "Recovery" macro-phase of the ASRS.
      - Sequences all sub-steps needed to recover sample from Andersen stages:
          1) Meter solvent 1
          2) Recirculate solvent 1
          3) Soak solvent
          4) Clean lines (solvent 1)
          5) (Optional) Meter solvent 2
          6) Agitate and mix solvents 1 & 2
          7) Clean lines (solvent 1 & 2)
          8) Prime needles
          9) Fill vials (rows 1–4, according to recipe)
         10) Waste remaining solvent
         11) Mark phase as completed

      - Updates HMI progress bar and status text during the entire phase.

    Usage:
      - Call cyclically with bExecute = TRUE while the machine is in
        the Recovery Phase state.
      - Internal state machine (eRecoveryState) will progress through
        each recovery step.
      - When eRecoveryState reaches "Completed", bSuccess = TRUE.

    Inputs:
      - bExecute : BOOL
          TRUE  → start/continue the recovery phase.
          FALSE → keeps FB in Idle (no progression).

    Outputs:
      - bSuccess : BOOL
          TRUE when the full recovery sequence finishes successfully.
      - bError   : BOOL
          TRUE if an error is detected in the recovery phase
          (hook for future error handling, currently not fully used).

    Side Effects:
      - Writes to global HMI animation:
          GVL_HMI.HMIAnimation.sLoadTextRecovery
          GVL_HMI.HMIAnimation.rLoadBarRecovery
          GVL_HMI.HMIAnimation.eIconStateRecovery
      - Uses global recipe/settings structures to decide which steps
        are required (number of solvents, vials to fill, etc.).
*)

FUNCTION_BLOCK FB_RecoveryPhase
VAR_INPUT
    bExecute : BOOL;  // TRUE to start/maintain the recovery phase
END_VAR

VAR_OUTPUT
    bSuccess : BOOL;  // Phase finished successfully
    bError   : BOOL;  // Phase error flag (reserved for future detailed handling)
END_VAR

VAR
    // -----------------------------
    // Internal Recovery FSM state
    // -----------------------------
    eRecoveryState : E_RecoveryState := E_RecoveryState.Idle;

    // -----------------------------
    // Sub-function blocks
    // -----------------------------
    fbSolenoidControl  : FB_SolenoidControl;  // Reserved: control of solenoid configuration
    fbMeteringSolvent1 : FB_MeteringSolvent1; // Reserved: specific metering FB (not used directly here)

    // -----------------------------
    // Error handling (reserved hooks)
    // -----------------------------
    bErrorDetected : BOOL := FALSE;   // TRUE if any error is detected internally
    nPumpWithError : INT := 0;        // Stores pump index that failed
    nErrorID       : UDINT := 0;      // Error code identifier (for diagnostics)

    // -----------------------------
    // Generic step / loop helpers
    // -----------------------------
    iStepCounter : INT := 0;   // Generic counter used in step subroutines
    i           : USINT;       // Generic loop index (for internal use)

    // -----------------------------
    // Control flags for movements
    // -----------------------------
    bStart             : BOOL := FALSE; // Local start latch derived from bExecute
    bMoveM2            : BOOL := FALSE; // Reserved: movement flag for Motor M2
    bMoveM3            : BOOL := FALSE; // Reserved: movement flag for Motor M3
    bMovementComplete  : BOOL := FALSE; // TRUE when the active sub-step has finished

    // -----------------------------
    // Metering control (solvent 1 & 2)
    // -----------------------------
    bMoveValveDone : ARRAY[1..5] OF BOOL;  // Flags for valve moves completion
    bMovePumpDone  : ARRAY[1..10] OF BOOL; // Flags for pump moves completion
    fDistance      : ARRAY[1..10] OF REAL; // Distances for pump movements (metering)

    // -----------------------------
    // Recirculation control
    // -----------------------------
    fAgitationTime     : REAL := 0.0;           // Time used for agitation
    fRecirculationTime : REAL := 0.0;           // Time used for recirculation
    fCalcDistance      : ARRAY[1..10] OF REAL;  // Calculated pump distances for recirculation

    // -----------------------------
    // Solvent soak timing
    // -----------------------------
    timerSoak      : TON;        // Soak timer (TON)
    bTimerStarted  : BOOL := FALSE;
    bSoakTimerDone : BOOL := FALSE;

    // -----------------------------
    // Agitation timers (solvent 1 and 2)
    // -----------------------------
    tonAgitateTime1 : TON;       // Timer for first agitation phase
    tonAgitateTime2 : TON;       // Timer for second agitation phase

    // -----------------------------
    // HMI Progress Bar Timing
    // -----------------------------
    rTotalEstimatedTimeSec : REAL := 0.0; // Estimated total duration of recovery phase (seconds)
    rElapsedTimeSec        : REAL := 0.0; // Elapsed time since start (seconds)
    tStartTime             : TIME := T#0S; // Time when recovery phase started
    bProgressInitDone      : BOOL := FALSE; // TRUE when progress timing has been initialized
END_VAR

// ==========================================================================
// 1) Start latch:
//    On first bExecute = TRUE, set bStart and put FSM into Idle.
// ==========================================================================
IF NOT bStart THEN
    eRecoveryState := E_RecoveryState.Idle;
    bStart         := bExecute; // Latch start when execution is requested
END_IF

// ==========================================================================
// 2) HMI progress bar update
//    - Only updates while FSM is actively running (not Idle/Completed)
//    - Uses rTotalEstimatedTimeSec from an external EstimateTotalTime() fn.
// ==========================================================================
IF bProgressInitDone
   AND (eRecoveryState <> E_RecoveryState.Idle)
   AND (eRecoveryState <> E_RecoveryState.Completed)
THEN
    // Compute elapsed time in seconds since recovery start
    rElapsedTimeSec := TO_REAL(TIME() - tStartTime) / 1000.0;

    // Scale 0..elapsed..total into a 0..100 % load bar
    // MIN() prevents overshoot in case of longer-than-expected duration.
    GVL_HMI.HMIAnimation.rLoadBarRecovery :=
        MIN(100.0, rElapsedTimeSec / rTotalEstimatedTimeSec * 100.0);
END_IF

// ==========================================================================
// 3) Recovery Phase FSM
// ==========================================================================
CASE eRecoveryState OF

    // ----------------------------------------------------------------------
    // Idle:
    //  - Waiting for bStart to be set.
    //  - Initializes HMI and timing once the phase starts.
    // ----------------------------------------------------------------------
    E_RecoveryState.Idle:

        bSuccess := FALSE;
        bError   := FALSE;

        IF bStart THEN
            // Initialize timing for progress bar
            tStartTime             := TIME();
            rTotalEstimatedTimeSec := EstimateTotalTime(); // External estimate
            bProgressInitDone      := TRUE;

            // Configure HMI animation for Recovery Phase start
            GVL_HMI.HMIAnimation.sLoadTextRecovery   := 'Starting';
            GVL_HMI.HMIAnimation.rLoadBarRecovery    := 0.0;
            GVL_HMI.HMIAnimation.eIconStateRecovery  := E_IconState.InProgress;

            // Move to first step: Metering of Solvent 1
            eRecoveryState := E_RecoveryState.Metering_Solvent1;
        END_IF;


    // ----------------------------------------------------------------------
    // Metering_Solvent1:
    //  - Meter solvent 1 into Andersen stages according to recipe.
    //  - If sealing+metering was already done in seal phase (flag),
    //    this step can be skipped.
    // ----------------------------------------------------------------------
    E_RecoveryState.Metering_Solvent1: // Could be replaced by external FB in parallel if needed

        // If general seal+pump already metered solvent 1, skip movement
        IF GVL_Settings.bGeneralSealAndPump
           AND GVL_Settings.bMeteringSolvent1Done
        THEN
            bMovementComplete := TRUE;
        ELSE
            // Execute local metering logic (subroutine)
            MeteringSolvent1();
        END_IF

        // On completion, go to recirculation with solvent 1
        IF bMovementComplete THEN
            eRecoveryState        := E_RecoveryState.Recirculate_Solvent1;
            iStepCounter          := 0;
            GVL_Settings.bMeteringSolvent1Done := FALSE;
            bMovementComplete     := FALSE;
        END_IF


    // ----------------------------------------------------------------------
    // Recirculate_Solvent1:
    //  - Recirculates solvent 1 to promote mixing and wetting of stages.
    // ----------------------------------------------------------------------
    E_RecoveryState.Recirculate_Solvent1:

        RecirculateSolvent1();

        IF bMovementComplete THEN
            eRecoveryState    := E_RecoveryState.Solvent_Soak;
            iStepCounter      := 0;
            bMovementComplete := FALSE;
        END_IF


    // ----------------------------------------------------------------------
    // Solvent_Soak:
    //  - Keeps solvent in contact with stages for a soak time (timer based).
    // ----------------------------------------------------------------------
    E_RecoveryState.Solvent_Soak:

        SolventSoak();

        IF bMovementComplete THEN
            eRecoveryState    := E_RecoveryState.Cleaning_Lines_S1;
            iStepCounter      := 0;
            bMovementComplete := FALSE;
        END_IF


    // ----------------------------------------------------------------------
    // Cleaning_Lines_S1:
    //  - Cleans fluidic lines used with solvent 1.
    //  - If recipe requires solvent 2 for recovery, proceed to its metering.
    //  - Otherwise, skip ahead to Prime_Needles.
    // ----------------------------------------------------------------------
    E_RecoveryState.Cleaning_Lines_S1:

        CleaningLinesSolvent1();

        IF bMovementComplete THEN
            // Check if solvent 2 is configured for recovery:
            // aSolventN[2] = 0 → second solvent not used.
            IF GVL_Recipe.stActiveRecipe.stSolventsTimes.aSolventN[2] <> 0 THEN
                eRecoveryState := E_RecoveryState.Metering_Solvent2;
            ELSE
                // Skip directly to needle priming if solvent 2 is not needed
                eRecoveryState := E_RecoveryState.Prime_Needles;
            END_IF

            iStepCounter      := 0;
            bMovementComplete := FALSE;
        END_IF


    // ----------------------------------------------------------------------
    // Metering_Solvent2:
    //  - Meters solvent 2, if configured, for recovery phase.
    // ----------------------------------------------------------------------
    E_RecoveryState.Metering_Solvent2:

        MeteringSolvent2();

        IF bMovementComplete THEN
            eRecoveryState    := E_RecoveryState.AgitateTime1;
            iStepCounter      := 0;
            bMovementComplete := FALSE;
        END_IF


    // ----------------------------------------------------------------------
    // AgitateTime1:
    //  - First agitation time window after solvent 2 metering.
    // ----------------------------------------------------------------------
    E_RecoveryState.AgitateTime1:

        AgitateTime1();

        IF bMovementComplete THEN
            eRecoveryState    := E_RecoveryState.Mix_Solvent1_2;
            iStepCounter      := 0;
            bMovementComplete := FALSE;
        END_IF


    // ----------------------------------------------------------------------
    // Mix_Solvent1_2:
    //  - Mixes solvents 1 and 2 inside Andersen stages or fluidic path.
    // ----------------------------------------------------------------------
    E_RecoveryState.Mix_Solvent1_2:

        MixSolvent1and2();

        IF bMovementComplete THEN
            eRecoveryState    := E_RecoveryState.Cleaning_Lines_S1_S2;
            iStepCounter      := 0;
            bMovementComplete := FALSE;
        END_IF


    // ----------------------------------------------------------------------
    // Cleaning_Lines_S1_S2:
    //  - Cleans all lines used for solvent 1 and solvent 2.
    // ----------------------------------------------------------------------
    E_RecoveryState.Cleaning_Lines_S1_S2:

